gfCNCPoint1[1221] = {X 523.1434, Y 21.1314, Z -1.3333, A 0.000, B 0.000, C 0.000 }
gfCNCPoint1[1222] = {X 523.9777, Y 20.6072, Z -1.3333, A 0.000, B 0.000, C 0.000 }
gfCNCPoint1[1223] = {X 524.9077, Y 20.2817, Z -1.3333, A 0.000, B 0.000, C 0.000 }
gfCNCPoint1[1224] = {X 525.8868, Y 20.1714, Z -1.3333, A 0.000, B 0.000, C 0.000 }
gfCNCPoint1[1225] = {X 526.5702, Y 20.1716, Z -1.3333, A 0.000, B 0.000, C 0.000 }
gfCNCPoint1[1226] = {X 527.4025, Y 20.2591, Z -1.3333, A 0.000, B 0.000, C 0.000 }
gfCNCPoint1[1227] = {X 528.2032, Y 20.5026, Z -1.3333, A 0.000, B 0.000, C 0.000 }
gfCNCPoint1[1228] = {X 528.9433, Y 20.8933, Z -1.3333, A 0.000, B 0.000, C 0.000 }
gfCNCPoint1[1229] = {X 529.5960, Y 21.4171, Z -1.3333, A 0.000, B 0.000, C 0.000 }
gfCNCPoint1[1230] = {X 530.1378, Y 22.0550, Z -1.3333, A 0.000, B 0.000, C 0.000 }
gfCNCPoint1[1231] = {X 534.5519, Y 22.0554, Z -1.3333, A 0.000, B 0.000, C 0.000 }
gfCNCPoint1[1232] = {X 534.5519, Y 19.7809, Z -1.3333, A 0.000, B 0.000, C 0.000 }
gfCNCPoint1[1233] = {X 528.8157, Y 19.7807, Z -1.3333, A 0.000, B 0.000, C 0.000 }
gfCNCPoint1[1234] = {X 528.8157, Y 20.2607, Z -1.3333, A 0.000, B 0.000, C 0.000 }
gfCNCPoint1[1235] = {X 534.0719, Y 20.2609, Z -1.3333, A 0.000, B 0.000, C 0.000 }
gfCNCPoint1[1236] = {X 534.0719, Y 21.5753, Z -1.3333, A 0.000, B 0.000, C 0.000 }
gfCNCPoint1[1237] = {X 530.3802, Y 21.5750, Z -1.3333, A 0.000, B 0.000, C 0.000 }
gfCNCPoint1[1238] = {X 529.6675, Y 20.8350, Z -1.3333, A 0.000, B 0.000, C 0.000 }
gfCNCPoint1[1239] = {X 528.8157, Y 20.2607, Z -1.3333, A 0.000, B 0.000, C 0.000 }
gfCNCPoint1[1240] = {X 528.8157, Y 19.7807, Z -1.3333, A 0.000, B 0.000, C 0.000 }
gfCNCPoint1[1241] = {X 524.2352, Y 19.7804, Z -1.3333, A 0.000, B 0.000, C 0.000 }
gfCNCPoint1[1242] = {X 523.6875, Y 20.4311, Z -1.3333, A 0.000, B 0.000, C 0.000 }
gfCNCPoint1[1243] = {X 523.0249, Y 20.9643, Z -1.3333, A 0.000, B 0.000, C 0.000 }
gfCNCPoint1[1244] = {X 522.2721, Y 21.3600, Z -1.3333, A 0.000, B 0.000, C 0.000 }
gfCNCPoint1[1245] = {X 521.4572, Y 21.6035, Z -1.3333, A 0.000, B 0.000, C 0.000 }
gfCNCPoint1[1246] = {X 520.6107, Y 21.6857, Z -1.3333, A 0.000, B 0.000, C 0.000 }
gfCNCPoint1[1247] = {X 519.9691, Y 21.6857, Z -1.3333, A 0.000, B 0.000, C 0.000 }
gfCNCPoint1[1248] = {X 518.9900, Y 21.5754, Z -1.3333, A 0.000, B 0.000, C 0.000 }
gfCNCPoint1[1249] = {X 518.0600, Y 21.2500, Z -1.3333, A 0.000, B 0.000, C 0.000 }
gfCNCPoint1[1250] = {X 517.2257, Y 20.7258, Z -1.3333, A 0.000, B 0.000, C 0.000 }
gfCNCPoint1[1251] = {X 516.5290, Y 20.0291, Z -1.3333, A 0.000, B 0.000, C 0.000 }
gfCNCPoint1[1252] = {X 516.0048, Y 19.1948, Z -1.3333, A 0.000, B 0.000, C 0.000 }
gfCNCPoint1[1253] = {X 515.6794, Y 18.2648, Z -1.3333, A 0.000, B 0.000, C 0.000 }
gfCNCPoint1[1254] = {X 515.5691, Y 17.2857, Z -1.3333, A 0.000, B 0.000, C 0.000 }
gfCNCPoint1[1255] = {X 515.5691, Y 10.3077, Z -1.3333, A 0.000, B 0.000, C 0.000 }
gfCNCPoint1[1256] = {X 515.6394, Y 9.5244, Z -1.3333, A 0.000, B 0.000, C 0.000 }
gfCNCPoint1[1257] = {X 515.8480, Y 8.7662, Z -1.3333, A 0.000, B 0.000, C 0.000 }
gfCNCPoint1[1258] = {X 516.1882, Y 8.0572, Z -1.3333, A 0.000, B 0.000, C 0.000 }
gfCNCPoint1[1259] = {X 516.6492, Y 7.4201, Z -1.3333, A 0.000, B 0.000, C 0.000 }
gfCNCPoint1[1260] = {X 516.2870, Y 7.1051, Z -1.3333, A 0.000, B 0.000, C 0.000 }
gfCNCPoint1[1261] = {X 469.2627, Y 7.1051, Z -1.3333, A 0.000, B 0.000, C 0.000 }
gfCNCPoint1[1262] = {X 469.2627, Y 11.9051, Z -1.3333, A 0.000, B 0.000, C 0.000 }
gfCNCPoint1[1263] = {X 469.1139, Y 11.9051, Z -1.3333, A 0.000, B 0.000, C 0.000 }
gfCNCPoint1[1264] = {X 469.1170, Y 12.0458, Z -1.3333, A 0.000, B 0.000, C 0.000 }
gfCNCPoint1[1265] = {X 469.1179, Y 12.1865, Z -1.3333, A 0.000, B 0.000, C 0.000 }
gfCNCPoint1[1266] = {X 469.1897, Y 12.0455, Z -1.3333, A 0.000, B 0.000, C 0.000 }
gfCNCPoint1[1267] = {X 469.2627, Y 11.9051, Z -1.3333, A 0.000, B 0.000, C 0.000 }
gfCNCPoint1[1268] = {X 469.2627, Y 9.5051, Z -1.3333, A 0.000, B 0.000, C 0.000 }
gfCNCPoint1[1269] = {X 466.2067, Y 9.5051, Z -1.3333, A 0.000, B 0.000, C 0.000 }
gfCNCPoint1[1270] = {X 466.5686, Y 10.7174, Z -1.3333, A 0.000, B 0.000, C 0.000 }
gfCNCPoint1[1271] = {X 466.7149, Y 11.9742, Z -1.3333, A 0.000, B 0.000, C 0.000 }
gfCNCPoint1[1272] = {X 466.7172, Y 12.0787, Z -1.3333, A 0.000, B 0.000, C 0.000 }
gfCNCPoint1[1273] = {X 466.7179, Y 12.1834, Z -1.3333, A 0.000, B 0.000, C 0.000 }
gfCNCPoint1[1274] = {X 466.7179, Y 12.9779, Z -1.3333, A 0.000, B 0.000, C 0.000 }
gfCNCPoint1[1275] = {X 466.6191, Y 14.1735, Z -1.3333, A 0.000, B 0.000, C 0.000 }
gfCNCPoint1[1276] = {X 466.3252, Y 15.3367, Z -1.3333, A 0.000, B 0.000, C 0.000 }
gfCNCPoint1[1277] = {X 465.8443, Y 16.4358, Z -1.3333, A 0.000, B 0.000, C 0.000 }
gfCNCPoint1[1278] = {X 465.1894, Y 17.4410, Z -1.3333, A 0.000, B 0.000, C 0.000 }
gfCNCPoint1[1279] = {X 465.1896, Y 25.8683, Z -1.3333, A 0.000, B 0.000, C 0.000 }
gfCNCPoint1[1280] = {X 467.5896, Y 25.8683, Z -1.3333, A 0.000, B 0.000, C 0.000 }
gfCNCPoint1[1281] = {X 467.5898, Y 38.9887, Z -1.3333, A 0.000, B 0.000, C 0.000 }
gfCNCPoint1[1282] = {X 467.6015, Y 39.0069, Z -1.3333, A 0.000, B 0.000, C 0.000 }
gfCNCPoint1[1283] = {X 468.3506, Y 37.9855, Z -1.3333, A 0.000, B 0.000, C 0.000 }
gfCNCPoint1[1284] = {X 469.2267, Y 37.0706, Z -1.3333, A 0.000, B 0.000, C 0.000 }
gfCNCPoint1[1285] = {X 470.2148, Y 36.2780, Z -1.3333, A 0.000, B 0.000, C 0.000 }
gfCNCPoint1[1286] = {X 471.5281, Y 33.7072, Z -1.3333, A 0.000, B 0.000, C 0.000 }
gfCNCPoint1[1287] = {X 470.4815, Y 32.4113, Z -1.3333, A 0.000, B 0.000, C 0.000 }
gfCNCPoint1[1288] = {X 469.5681, Y 31.0183, Z -1.3333, A 0.000, B 0.000, C 0.000 }
gfCNCPoint1[1289] = {X 468.7969, Y 29.5419, Z -1.3333, A 0.000, B 0.000, C 0.000 }
gfCNCPoint1[1290] = {X 468.1754, Y 27.9964, Z -1.3333, A 0.000, B 0.000, C 0.000 }
gfCNCPoint1[1291] = {X 467.7096, Y 26.3971, Z -1.3333, A 0.000, B 0.000, C 0.000 }
gfCNCPoint1[1292] = {X 467.6480, Y 26.1331, Z -1.3333, A 0.000, B 0.000, C 0.000 }
gfCNCPoint1[1293] = {X 467.5896, Y 25.8683, Z -1.3333, A 0.000, B 0.000, C 0.000 }
gfCNCPoint1[1294] = {X 465.1896, Y 25.8683, Z -1.3333, A 0.000, B 0.000, C 0.000 }
gfCNCPoint1[1295] = {X 465.1898, Y 39.7463, Z -1.3333, A 0.000, B 0.000, C 0.000 }
gfCNCPoint1[1296] = {X 465.3900, Y 40.0170, Z -1.3333, A 0.000, B 0.000, C 0.000 }
gfCNCPoint1[1297] = {X 465.5774, Y 40.2966, Z -1.3333, A 0.000, B 0.000, C 0.000 }
gfCNCPoint1[1298] = {X 466.0634, Y 41.1919, Z -1.3333, A 0.000, B 0.000, C 0.000 }
gfCNCPoint1[1299] = {X 466.4196, Y 42.1462, Z -1.3333, A 0.000, B 0.000, C 0.000 }
gfCNCPoint1[1300] = {X 466.6392, Y 43.1408, Z -1.3333, A 0.000, B 0.000, C 0.000 }
gfCNCPoint1[1301] = {X 466.7178, Y 44.1564, Z -1.3333, A 0.000, B 0.000, C 0.000 }
gfCNCPoint1[1302] = {X 466.7179, Y 45.0000, Z -1.3333, A 0.000, B 0.000, C 0.000 }
gfCNCPoint1[1303] = {X 466.7033, Y 45.4609, Z -1.3333, A 0.000, B 0.000, C 0.000 }
gfCNCPoint1[1304] = {X 466.6596, Y 45.9200, Z -1.3333, A 0.000, B 0.000, C 0.000 }
gfCNCPoint1[1305] = {X 468.5433, Y 45.9200, Z -1.3333, A 0.000, B 0.000, C 0.000 }
gfCNCPoint1[1306] = {X 468.4996, Y 45.4609, Z -1.3333, A 0.000, B 0.000, C 0.000 }
gfCNCPoint1[1307] = {X 468.4850, Y 45.0000, Z -1.3333, A 0.000, B 0.000, C 0.000 }
gfCNCPoint1[1308] = {X 468.4850, Y 44.2090, Z -1.3333, A 0.000, B 0.000, C 0.000 }
gfCNCPoint1[1309] = {X 468.5580, Y 43.1799, Z -1.3333, A 0.000, B 0.000, C 0.000 }
gfCNCPoint1[1310] = {X 468.7759, Y 42.1714, Z -1.3333, A 0.000, B 0.000, C 0.000 }
gfCNCPoint1[1311] = {X 469.1341, Y 41.2038, Z -1.3333, A 0.000, B 0.000, C 0.000 }
gfCNCPoint1[1312] = {X 469.6255, Y 40.2966, Z -1.3333, A 0.000, B 0.000, C 0.000 }
gfCNCPoint1[1313] = {X 470.3102, Y 39.3876, Z -1.3333, A 0.000, B 0.000, C 0.000 }
gfCNCPoint1[1314] = {X 471.1282, Y 38.5964, Z -1.3333, A 0.000, B 0.000, C 0.000 }
gfCNCPoint1[1315] = {X 472.0595, Y 37.9424, Z -1.3333, A 0.000, B 0.000, C 0.000 }
gfCNCPoint1[1316] = {X 474.4573, Y 33.2490, Z -1.3333, A 0.000, B 0.000, C 0.000 }
gfCNCPoint1[1317] = {X 473.2262, Y 32.0044, Z -1.3333, A 0.000, B 0.000, C 0.000 }
gfCNCPoint1[1318] = {X 472.1548, Y 30.6199, Z -1.3333, A 0.000, B 0.000, C 0.000 }
gfCNCPoint1[1319] = {X 471.2590, Y 29.1158, Z -1.3333, A 0.000, B 0.000, C 0.000 }
gfCNCPoint1[1320] = {X 470.5519, Y 27.5144, Z -1.3333, A 0.000, B 0.000, C 0.000 }
gfCNCPoint1[1321] = {X 470.0438, Y 25.8391, Z -1.3333, A 0.000, B 0.000, C 0.000 }
gfCNCPoint1[1322] = {X 469.9887, Y 25.6028, Z -1.3333, A 0.000, B 0.000, C 0.000 }
gfCNCPoint1[1323] = {X 469.9364, Y 25.3658, Z -1.3333, A 0.000, B 0.000, C 0.000 }
gfCNCPoint1[1324] = {X 469.6267, Y 23.4734, Z -1.3333, A 0.000, B 0.000, C 0.000 }
gfCNCPoint1[1325] = {X 469.5026, Y 21.5599, Z -1.3333, A 0.000, B 0.000, C 0.000 }
gfCNCPoint1[1326] = {X 469.5653, Y 19.6434, Z -1.3333, A 0.000, B 0.000, C 0.000 }
gfCNCPoint1[1327] = {X 469.8141, Y 17.7420, Z -1.3333, A 0.000, B 0.000, C 0.000 }
gfCNCPoint1[1328] = {X 470.2468, Y 15.8739, Z -1.3333, A 0.000, B 0.000, C 0.000 }
gfCNCPoint1[1329] = {X 470.6926, Y 14.5452, Z -1.3333, A 0.000, B 0.000, C 0.000 }
gfCNCPoint1[1330] = {X 471.2622, Y 13.2646, Z -1.3333, A 0.000, B 0.000, C 0.000 }
gfCNCPoint1[1331] = {X 471.3239, Y 13.1432, Z -1.3333, A 0.000, B 0.000, C 0.000 }
gfCNCPoint1[1332] = {X 471.3867, Y 13.0225, Z -1.3333, A 0.000, B 0.000, C 0.000 }
gfCNCPoint1[1333] = {X 472.1282, Y 11.7671, Z -1.3333, A 0.000, B 0.000, C 0.000 }
gfCNCPoint1[1334] = {X 472.9897, Y 10.5909, Z -1.3333, A 0.000, B 0.000, C 0.000 }
gfCNCPoint1[1335] = {X 473.9628, Y 9.5051, Z -1.3333, A 0.000, B 0.000, C 0.000 }
gfCNCPoint1[1336] = {X 469.2627, Y 9.5051, Z -1.3333, A 0.000, B 0.000, C 0.000 }
gfCNCPoint1[1337] = {X 469.2627, Y 7.1051, Z -1.3333, A 0.000, B 0.000, C 0.000 }
gfCNCPoint1[1338] = {X 370.1016, Y 7.1051, Z -1.3333, A 0.000, B 0.000, C 0.000 }
gfCNCPoint1[1339] = {X 371.1252, Y 8.7921, Z -1.3333, A 0.000, B 0.000, C 0.000 }
gfCNCPoint1[1340] = {X 372.0361, Y 10.5425, Z -1.3333, A 0.000, B 0.000, C 0.000 }
gfCNCPoint1[1341] = {X 372.9332, Y 12.6093, Z -1.3333, A 0.000, B 0.000, C 0.000 }
gfCNCPoint1[1342] = {X 373.6731, Y 14.7374, Z -1.3333, A 0.000, B 0.000, C 0.000 }
gfCNCPoint1[1343] = {X 374.2517, Y 16.9150, Z -1.3333, A 0.000, B 0.000, C 0.000 }
gfCNCPoint1[1344] = {X 374.7361, Y 19.4755, Z -1.3333, A 0.000, B 0.000, C 0.000 }
gfCNCPoint1[1345] = {X 375.0392, Y 22.0637, Z -1.3333, A 0.000, B 0.000, C 0.000 }
gfCNCPoint1[1346] = {X 375.1593, Y 24.6669, Z -1.3333, A 0.000, B 0.000, C 0.000 }
gfCNCPoint1[1347] = {X 375.0959, Y 27.2721, Z -1.3333, A 0.000, B 0.000, C 0.000 }
gfCNCPoint1[1348] = {X 374.8493, Y 29.8664, Z -1.3333, A 0.000, B 0.000, C 0.000 }
gfCNCPoint1[1349] = {X 374.4207, Y 32.4368, Z -1.3333, A 0.000, B 0.000, C 0.000 }
gfCNCPoint1[1350] = {X 373.7829, Y 34.9988, Z -1.3333, A 0.000, B 0.000, C 0.000 }
gfCNCPoint1[1351] = {X 372.9214, Y 37.4945, Z -1.3333, A 0.000, B 0.000, C 0.000 }
gfCNCPoint1[1352] = {X 371.8430, Y 39.9043, Z -1.3333, A 0.000, B 0.000, C 0.000 }
gfCNCPoint1[1353] = {X 370.5559, Y 42.2095, Z -1.3333, A 0.000, B 0.000, C 0.000 }
gfCNCPoint1[1354] = {X 369.0704, Y 44.3921, Z -1.3333, A 0.000, B 0.000, C 0.000 }
gfCNCPoint1[1355] = {X 369.0316, Y 44.4442, Z -1.3333, A 0.000, B 0.000, C 0.000 }
gfCNCPoint1[1356] = {X 368.9927, Y 44.4963, Z -1.3333, A 0.000, B 0.000, C 0.000 }
gfCNCPoint1[1357] = {X 367.4727, Y 46.3512, Z -1.3333, A 0.000, B 0.000, C 0.000 }
gfCNCPoint1[1358] = {X 365.7972, Y 48.0668, Z -1.3333, A 0.000, B 0.000, C 0.000 }
gfCNCPoint1[1359] = {X 363.9787, Y 49.6301, Z -1.3333, A 0.000, B 0.000, C 0.000 }
gfCNCPoint1[1360] = {X 362.0311, Y 51.0293, Z -1.3333, A 0.000, B 0.000, C 0.000 }
gfCNCPoint1[1361] = {X 359.9692, Y 52.2538, Z -1.3333, A 0.000, B 0.000, C 0.000 }
gfCNCPoint1[1362] = {X 359.3965, Y 52.5409, Z -1.3333, A 0.000, B 0.000, C 0.000 }
gfCNCPoint1[1363] = {X 358.8175, Y 52.8148, Z -1.3333, A 0.000, B 0.000, C 0.000 }
gfCNCPoint1[1364] = {X 356.4598, Y 53.7700, Z -1.3333, A 0.000, B 0.000, C 0.000 }
gfCNCPoint1[1365] = {X 354.0251, Y 54.5072, Z -1.3333, A 0.000, B 0.000, C 0.000 }
gfCNCPoint1[1366] = {X 351.5336, Y 55.0204, Z -1.3333, A 0.000, B 0.000, C 0.000 }
gfCNCPoint1[1367] = {X 349.0058, Y 55.3053, Z -1.3333, A 0.000, B 0.000, C 0.000 }
gfCNCPoint1[1368] = {X 349.9666, Y 69.6732, Z -1.3333, A 0.000, B 0.000, C 0.000 }
gfCNCPoint1[1369] = {X 348.6526, Y 69.7406, Z -1.3333, A 0.000, B 0.000, C 0.000 }
gfCNCPoint1[1370] = {X 347.3372, Y 69.7672, Z -1.3333, A 0.000, B 0.000, C 0.000 }
gfCNCPoint1[1371] = {X 346.5718, Y 69.7758, Z -1.3333, A 0.000, B 0.000, C 0.000 }
gfCNCPoint1[1372] = {X 345.8063, Y 69.7711, Z -1.3333, A 0.000, B 0.000, C 0.000 }
gfCNCPoint1[1373] = {X 345.5910, Y 70.1878, Z -1.3333, A 0.000, B 0.000, C 0.000 }
gfCNCPoint1[1374] = {X 345.3676, Y 70.6003, Z -1.3333, A 0.000, B 0.000, C 0.000 }
gfCNCPoint1[1375] = {X 345.9399, Y 70.6040, Z -1.3333, A 0.000, B 0.000, C 0.000 }
gfCNCPoint1[1376] = {X 348.1990, Y 70.6282, Z -1.3333, A 0.000, B 0.000, C 0.000 }
gfCNCPoint1[1377] = {X 350.4581, Y 70.6078, Z -1.3333, A 0.000, B 0.000, C 0.000 }
gfCNCPoint1[1378] = {X 350.2072, Y 70.1432, Z -1.3333, A 0.000, B 0.000, C 0.000 }
gfCNCPoint1[1379] = {X 349.9666, Y 69.6732, Z -1.3333, A 0.000, B 0.000, C 0.000 }
gfCNCPoint1[1380] = {X 349.8065, Y 67.2785, Z -1.3333, A 0.000, B 0.000, C 0.000 }
gfCNCPoint1[1381] = {X 348.5577, Y 67.3424, Z -1.3333, A 0.000, B 0.000, C 0.000 }
gfCNCPoint1[1382] = {X 347.3075, Y 67.3673, Z -1.3333, A 0.000, B 0.000, C 0.000 }
gfCNCPoint1[1383] = {X 345.8014, Y 67.3707, Z -1.3333, A 0.000, B 0.000, C 0.000 }
gfCNCPoint1[1384] = {X 344.2963, Y 67.3191, Z -1.3333, A 0.000, B 0.000, C 0.000 }
gfCNCPoint1[1385] = {X 343.8111, Y 68.3919, Z -1.3333, A 0.000, B 0.000, C 0.000 }
gfCNCPoint1[1386] = {X 343.2685, Y 69.4370, Z -1.3333, A 0.000, B 0.000, C 0.000 }
gfCNCPoint1[1387] = {X 342.7876, Y 70.2613, Z -1.3333, A 0.000, B 0.000, C 0.000 }
gfCNCPoint1[1388] = {X 342.2711, Y 71.0637, Z -1.3333, A 0.000, B 0.000, C 0.000 }
gfCNCPoint1[1389] = {X 342.2712, Y 72.9213, Z -1.3333, A 0.000, B 0.000, C 0.000 }
gfCNCPoint1[1390] = {X 343.8076, Y 72.9731, Z -1.3333, A 0.000, B 0.000, C 0.000 }
gfCNCPoint1[1391] = {X 345.3447, Y 73.0002, Z -1.3333, A 0.000, B 0.000, C 0.000 }
gfCNCPoint1[1392] = {X 345.6279, Y 73.0025, Z -1.3333, A 0.000, B 0.000, C 0.000 }
gfCNCPoint1[1393] = {X 345.9111, Y 73.0039, Z -1.3333, A 0.000, B 0.000, C 0.000 }
gfCNCPoint1[1394] = {X 348.2072, Y 73.0282, Z -1.3333, A 0.000, B 0.000, C 0.000 }
gfCNCPoint1[1395] = {X 350.5035, Y 73.0073, Z -1.3333, A 0.000, B 0.000, C 0.000 }
gfCNCPoint1[1396] = {X 352.0323, Y 72.9685, Z -1.3333, A 0.000, B 0.000, C 0.000 }
gfCNCPoint1[1397] = {X 353.5605, Y 72.9096, Z -1.3333, A 0.000, B 0.000, C 0.000 }
gfCNCPoint1[1398] = {X 353.5603, Y 71.0790, Z -1.3333, A 0.000, B 0.000, C 0.000 }
gfCNCPoint1[1399] = {X 353.0407, Y 70.2727, Z -1.3333, A 0.000, B 0.000, C 0.000 }
gfCNCPoint1[1400] = {X 352.5573, Y 69.4443, Z -1.3333, A 0.000, B 0.000, C 0.000 }
gfCNCPoint1[1401] = {X 351.9695, Y 68.3058, Z -1.3333, A 0.000, B 0.000, C 0.000 }
gfCNCPoint1[1402] = {X 351.4500, Y 67.1345, Z -1.3333, A 0.000, B 0.000, C 0.000 }
gfCNCPoint1[1403] = {X 350.6290, Y 67.2150, Z -1.3333, A 0.000, B 0.000, C 0.000 }
gfCNCPoint1[1404] = {X 349.8065, Y 67.2785, Z -1.3333, A 0.000, B 0.000, C 0.000 }
gfCNCPoint1[1405] = {X 349.6463, Y 64.8839, Z -1.3333, A 0.000, B 0.000, C 0.000 }
gfCNCPoint1[1406] = {X 348.4627, Y 64.9443, Z -1.3333, A 0.000, B 0.000, C 0.000 }
gfCNCPoint1[1407] = {X 347.2777, Y 64.9674, Z -1.3333, A 0.000, B 0.000, C 0.000 }
gfCNCPoint1[1408] = {X 344.9730, Y 64.9474, Z -1.3333, A 0.000, B 0.000, C 0.000 }
gfCNCPoint1[1409] = {X 342.6736, Y 64.7906, Z -1.3333, A 0.000, B 0.000, C 0.000 }
gfCNCPoint1[1410] = {X 341.9387, Y 66.7258, Z -1.3333, A 0.000, B 0.000, C 0.000 }
gfCNCPoint1[1411] = {X 341.0009, Y 68.5712, Z -1.3333, A 0.000, B 0.000, C 0.000 }
gfCNCPoint1[1412] = {X 339.8710, Y 70.3057, Z -1.3333, A 0.000, B 0.000, C 0.000 }
gfCNCPoint1[1413] = {X 339.8714, Y 75.1959, Z -1.3333, A 0.000, B 0.000, C 0.000 }
gfCNCPoint1[1414] = {X 342.8752, Y 75.3461, Z -1.3333, A 0.000, B 0.000, C 0.000 }
gfCNCPoint1[1415] = {X 345.8822, Y 75.4038, Z -1.3333, A 0.000, B 0.000, C 0.000 }
gfCNCPoint1[1416] = {X 350.9238, Y 75.3992, Z -1.3333, A 0.000, B 0.000, C 0.000 }
gfCNCPoint1[1417] = {X 355.9607, Y 75.1818, Z -1.3333, A 0.000, B 0.000, C 0.000 }
gfCNCPoint1[1418] = {X 355.9603, Y 70.3198, Z -1.3333, A 0.000, B 0.000, C 0.000 }
gfCNCPoint1[1419] = {X 355.0524, Y 68.9620, Z -1.3333, A 0.000, B 0.000, C 0.000 }
gfCNCPoint1[1420] = {X 354.2627, Y 67.5323, Z -1.3333, A 0.000, B 0.000, C 0.000 }
gfCNCPoint1[1421] = {X 353.5969, Y 66.0408, Z -1.3333, A 0.000, B 0.000, C 0.000 }
gfCNCPoint1[1422] = {X 353.0597, Y 64.4983, Z -1.3333, A 0.000, B 0.000, C 0.000 }
gfCNCPoint1[1423] = {X 351.3574, Y 64.7301, Z -1.3333, A 0.000, B 0.000, C 0.000 }
gfCNCPoint1[1424] = {X 349.6463, Y 64.8839, Z -1.3333, A 0.000, B 0.000, C 0.000 }
gfCNCPoint1[1425] = {X 349.4862, Y 62.4892, Z -1.3333, A 0.000, B 0.000, C 0.000 }
gfCNCPoint1[1426] = {X 348.3677, Y 62.5461, Z -1.3333, A 0.000, B 0.000, C 0.000 }
gfCNCPoint1[1427] = {X 347.2480, Y 62.5675, Z -1.3333, A 0.000, B 0.000, C 0.000 }
gfCNCPoint1[1428] = {X 345.1177, Y 62.5512, Z -1.3333, A 0.000, B 0.000, C 0.000 }
gfCNCPoint1[1429] = {X 342.9921, Y 62.4102, Z -1.3333, A 0.000, B 0.000, C 0.000 }
gfCNCPoint1[1430] = {X 340.8784, Y 62.1450, Z -1.3333, A 0.000, B 0.000, C 0.000 }
gfCNCPoint1[1431] = {X 340.4884, Y 63.7331, Z -1.3333, A 0.000, B 0.000, C 0.000 }
gfCNCPoint1[1432] = {X 339.9469, Y 65.2761, Z -1.3333, A 0.000, B 0.000, C 0.000 }
gfCNCPoint1[1433] = {X 339.2590, Y 66.7596, Z -1.3333, A 0.000, B 0.000, C 0.000 }
gfCNCPoint1[1434] = {X 338.4311, Y 68.1698, Z -1.3333, A 0.000, B 0.000, C 0.000 }
gfCNCPoint1[1435] = {X 337.4710, Y 69.4935, Z -1.3333, A 0.000, B 0.000, C 0.000 }
gfCNCPoint1[1436] = {X 337.4715, Y 77.4188, Z -1.3333, A 0.000, B 0.000, C 0.000 }
gfCNCPoint1[1437] = {X 341.6584, Y 77.6990, Z -1.3333, A 0.000, B 0.000, C 0.000 }
gfCNCPoint1[1438] = {X 345.8533, Y 77.8037, Z -1.3333, A 0.000, B 0.000, C 0.000 }
gfCNCPoint1[1439] = {X 350.0262, Y 77.8159, Z -1.3333, A 0.000, B 0.000, C 0.000 }
gfCNCPoint1[1440] = {X 354.1970, Y 77.6851, Z -1.3333, A 0.000, B 0.000, C 0.000 }
gfCNCPoint1[1441] = {X 358.3609, Y 77.4115, Z -1.3333, A 0.000, B 0.000, C 0.000 }
gfCNCPoint1[1442] = {X 358.3602, Y 69.5063, Z -1.3333, A 0.000, B 0.000, C 0.000 }
gfCNCPoint1[1443] = {X 357.3489, Y 68.1066, Z -1.3333, A 0.000, B 0.000, C 0.000 }
gfCNCPoint1[1444] = {X 356.4859, Y 66.6108, Z -1.3333, A 0.000, B 0.000, C 0.000 }
gfCNCPoint1[1445] = {X 355.7802, Y 65.0347, Z -1.3333, A 0.000, B 0.000, C 0.000 }
gfCNCPoint1[1446] = {X 355.2393, Y 63.3947, Z -1.3333, A 0.000, B 0.000, C 0.000 }
gfCNCPoint1[1447] = {X 354.8688, Y 61.7081, Z -1.3333, A 0.000, B 0.000, C 0.000 }
gfCNCPoint1[1448] = {X 352.1926, Y 62.2028, Z -1.3333, A 0.000, B 0.000, C 0.000 }
gfCNCPoint1[1449] = {X 349.4862, Y 62.4892, Z -1.3333, A 0.000, B 0.000, C 0.000 }
gfCNCPoint1[1450] = {X 349.3260, Y 60.0946, Z -1.3333, A 0.000, B 0.000, C 0.000 }
gfCNCPoint1[1451] = {X 348.2727, Y 60.1480, Z -1.3333, A 0.000, B 0.000, C 0.000 }
gfCNCPoint1[1452] = {X 347.2182, Y 60.1675, Z -1.3333, A 0.000, B 0.000, C 0.000 }
gfCNCPoint1[1453] = {X 344.3864, Y 60.1126, Z -1.3333, A 0.000, B 0.000, C 0.000 }
gfCNCPoint1[1454] = {X 341.5690, Y 59.8219, Z -1.3333, A 0.000, B 0.000, C 0.000 }
gfCNCPoint1[1455] = {X 338.7855, Y 59.2975, Z -1.3333, A 0.000, B 0.000, C 0.000 }
gfCNCPoint1[1456] = {X 338.6398, Y 60.9970, Z -1.3333, A 0.000, B 0.000, C 0.000 }
gfCNCPoint1[1457] = {X 338.2957, Y 62.6677, Z -1.3333, A 0.000, B 0.000, C 0.000 }
gfCNCPoint1[1458] = {X 337.7581, Y 64.2865, Z -1.3333, A 0.000, B 0.000, C 0.000 }
gfCNCPoint1[1459] = {X 337.0344, Y 65.8310, Z -1.3333, A 0.000, B 0.000, C 0.000 }
gfCNCPoint1[1460] = {X 336.1345, Y 67.2801, Z -1.3333, A 0.000, B 0.000, C 0.000 }
gfCNCPoint1[1461] = {X 335.0709, Y 68.6136, Z -1.3333, A 0.000, B 0.000, C 0.000 }
gfCNCPoint1[1462] = {X 335.0717, Y 79.5892, Z -1.3333, A 0.000, B 0.000, C 0.000 }
gfCNCPoint1[1463] = {X 335.6784, Y 79.6597, Z -1.3333, A 0.000, B 0.000, C 0.000 }
gfCNCPoint1[1464] = {X 336.2864, Y 79.7191, Z -1.3333, A 0.000, B 0.000, C 0.000 }
gfCNCPoint1[1465] = {X 341.0497, Y 80.0723, Z -1.3333, A 0.000, B 0.000, C 0.000 }
gfCNCPoint1[1466] = {X 345.8244, Y 80.2036, Z -1.3333, A 0.000, B 0.000, C 0.000 }
gfCNCPoint1[1467] = {X 350.3389, Y 80.2114, Z -1.3333, A 0.000, B 0.000, C 0.000 }
gfCNCPoint1[1468] = {X 354.8507, Y 80.0550, Z -1.3333, A 0.000, B 0.000, C 0.000 }
gfCNCPoint1[1469] = {X 359.3538, Y 79.7348, Z -1.3333, A 0.000, B 0.000, C 0.000 }
gfCNCPoint1[1470] = {X 360.0583, Y 79.6699, Z -1.3333, A 0.000, B 0.000, C 0.000 }
gfCNCPoint1[1471] = {X 360.7611, Y 79.5886, Z -1.3333, A 0.000, B 0.000, C 0.000 }
gfCNCPoint1[1472] = {X 360.7601, Y 68.6248, Z -1.3333, A 0.000, B 0.000, C 0.000 }
gfCNCPoint1[1473] = {X 359.7308, Y 67.3425, Z -1.3333, A 0.000, B 0.000, C 0.000 }
gfCNCPoint1[1474] = {X 358.8534, Y 65.9517, Z -1.3333, A 0.000, B 0.000, C 0.000 }
gfCNCPoint1[1475] = {X 358.1395, Y 64.4704, Z -1.3333, A 0.000, B 0.000, C 0.000 }
gfCNCPoint1[1476] = {X 357.5980, Y 62.9177, Z -1.3333, A 0.000, B 0.000, C 0.000 }
gfCNCPoint1[1477] = {X 357.2361, Y 61.3136, Z -1.3333, A 0.000, B 0.000, C 0.000 }
gfCNCPoint1[1478] = {X 357.0916, Y 60.1644, Z -1.3333, A 0.000, B 0.000, C 0.000 }
gfCNCPoint1[1479] = {X 357.0395, Y 59.0073, Z -1.3333, A 0.000, B 0.000, C 0.000 }
gfCNCPoint1[1480] = {X 357.0394, Y 58.6372, Z -1.3333, A 0.000, B 0.000, C 0.000 }
gfCNCPoint1[1481] = {X 355.6983, Y 59.0307, Z -1.3333, A 0.000, B 0.000, C 0.000 }
gfCNCPoint1[1482] = {X 354.3416, Y 59.3667, Z -1.3333, A 0.000, B 0.000, C 0.000 }
gfCNCPoint1[1483] = {X 351.8479, Y 59.8276, Z -1.3333, A 0.000, B 0.000, C 0.000 }
gfCNCPoint1[1484] = {X 349.3260, Y 60.0946, Z -1.3333, A 0.000, B 0.000, C 0.000 }
gfCNCPoint1[1485] = {X 349.1659, Y 57.6999, Z -1.3333, A 0.000, B 0.000, C 0.000 }
gfCNCPoint1[1486] = {X 348.1778, Y 57.7498, Z -1.3333, A 0.000, B 0.000, C 0.000 }
gfCNCPoint1[1487] = {X 347.1886, Y 57.7676, Z -1.3333, A 0.000, B 0.000, C 0.000 }
gfCNCPoint1[1488] = {X 344.5488, Y 57.7180, Z -1.3333, A 0.000, B 0.000, C 0.000 }
gfCNCPoint1[1489] = {X 341.9225, Y 57.4481, Z -1.3333, A 0.000, B 0.000, C 0.000 }
gfCNCPoint1[1490] = {X 339.3279, Y 56.9596, Z -1.3333, A 0.000, B 0.000, C 0.000 }
gfCNCPoint1[1491] = {X 337.7707, Y 56.5563, Z -1.3333, A 0.000, B 0.000, C 0.000 }
gfCNCPoint1[1492] = {X 336.2362, Y 56.0743, Z -1.3333, A 0.000, B 0.000, C 0.000 }
gfCNCPoint1[1493] = {X 336.3520, Y 57.0340, Z -1.3333, A 0.000, B 0.000, C 0.000 }
gfCNCPoint1[1494] = {X 336.3907, Y 58.0000, Z -1.3333, A 0.000, B 0.000, C 0.000 }
gfCNCPoint1[1495] = {X 336.3907, Y 58.9501, Z -1.3333, A 0.000, B 0.000, C 0.000 }
gfCNCPoint1[1496] = {X 336.3894, Y 59.0917, Z -1.3333, A 0.000, B 0.000, C 0.000 }
gfCNCPoint1[1497] = {X 336.3864, Y 59.2332, Z -1.3333, A 0.000, B 0.000, C 0.000 }
gfCNCPoint1[1498] = {X 336.2426, Y 60.7976, Z -1.3333, A 0.000, B 0.000, C 0.000 }
gfCNCPoint1[1499] = {X 335.8977, Y 62.3303, Z -1.3333, A 0.000, B 0.000, C 0.000 }
gfCNCPoint1[1500] = {X 335.3575, Y 63.8054, Z -1.3333, A 0.000, B 0.000, C 0.000 }
gfCNCPoint1[1501] = {X 334.6310, Y 65.1983, Z -1.3333, A 0.000, B 0.000, C 0.000 }
gfCNCPoint1[1502] = {X 333.7304, Y 66.4856, Z -1.3333, A 0.000, B 0.000, C 0.000 }
gfCNCPoint1[1503] = {X 332.6709, Y 67.6455, Z -1.3333, A 0.000, B 0.000, C 0.000 }
gfCNCPoint1[1504] = {X 332.6718, Y 81.6429, Z -1.3333, A 0.000, B 0.000, C 0.000 }
gfCNCPoint1[1505] = {X 334.3622, Y 81.9165, Z -1.3333, A 0.000, B 0.000, C 0.000 }
gfCNCPoint1[1506] = {X 336.0639, Y 82.1088, Z -1.3333, A 0.000, B 0.000, C 0.000 }
gfCNCPoint1[1507] = {X 340.9239, Y 82.4690, Z -1.3333, A 0.000, B 0.000, C 0.000 }
gfCNCPoint1[1508] = {X 345.7954, Y 82.6035, Z -1.3333, A 0.000, B 0.000, C 0.000 }
gfCNCPoint1[1509] = {X 350.3874, Y 82.6109, Z -1.3333, A 0.000, B 0.000, C 0.000 }
gfCNCPoint1[1510] = {X 354.9766, Y 82.4517, Z -1.3333, A 0.000, B 0.000, C 0.000 }
gfCNCPoint1[1511] = {X 359.5570, Y 82.1262, Z -1.3333, A 0.000, B 0.000, C 0.000 }
gfCNCPoint1[1512] = {X 361.3660, Y 81.9295, Z -1.3333, A 0.000, B 0.000, C 0.000 }
gfCNCPoint1[1513] = {X 363.1612, Y 81.6323, Z -1.3333, A 0.000, B 0.000, C 0.000 }
gfCNCPoint1[1514] = {X 363.1600, Y 67.6547, Z -1.3333, A 0.000, B 0.000, C 0.000 }
gfCNCPoint1[1515] = {X 362.0736, Y 66.4644, Z -1.3333, A 0.000, B 0.000, C 0.000 }
gfCNCPoint1[1516] = {X 361.1553, Y 65.1400, Z -1.3333, A 0.000, B 0.000, C 0.000 }
gfCNCPoint1[1517] = {X 360.4214, Y 63.7052, Z -1.3333, A 0.000, B 0.000, C 0.000 }
gfCNCPoint1[1518] = {X 359.8851, Y 62.1855, Z -1.3333, A 0.000, B 0.000, C 0.000 }
gfCNCPoint1[1519] = {X 359.5558, Y 60.6079, Z -1.3333, A 0.000, B 0.000, C 0.000 }
gfCNCPoint1[1520] = {X 359.4395, Y 59.0005, Z -1.3333, A 0.000, B 0.000, C 0.000 }
gfCNCPoint1[1521] = {X 359.4393, Y 58.0000, Z -1.3333, A 0.000, B 0.000, C 0.000 }
gfCNCPoint1[1522] = {X 359.5345, Y 56.4860, Z -1.3333, A 0.000, B 0.000, C 0.000 }
gfCNCPoint1[1523] = {X 359.8188, Y 54.9959, Z -1.3333, A 0.000, B 0.000, C 0.000 }
gfCNCPoint1[1524] = {X 358.0877, Y 55.7267, Z -1.3333, A 0.000, B 0.000, C 0.000 }
gfCNCPoint1[1525] = {X 356.3148, Y 56.3492, Z -1.3333, A 0.000, B 0.000, C 0.000 }
gfCNCPoint1[1526] = {X 353.9704, Y 56.9897, Z -1.3333, A 0.000, B 0.000, C 0.000 }
gfCNCPoint1[1527] = {X 351.5824, Y 57.4409, Z -1.3333, A 0.000, B 0.000, C 0.000 }
gfCNCPoint1[1528] = {X 349.1659, Y 57.6999, Z -1.3333, A 0.000, B 0.000, C 0.000 }
gfCNCPoint1[1529] = {X 349.0058, Y 55.3053, Z -1.3333, A 0.000, B 0.000, C 0.000 }
gfCNCPoint1[1530] = {X 348.0829, Y 55.3517, Z -1.3333, A 0.000, B 0.000, C 0.000 }
gfCNCPoint1[1531] = {X 347.1589, Y 55.3676, Z -1.3333, A 0.000, B 0.000, C 0.000 }
gfCNCPoint1[1532] = {X 344.5805, Y 55.3153, Z -1.3333, A 0.000, B 0.000, C 0.000 }
gfCNCPoint1[1533] = {X 342.0169, Y 55.0355, Z -1.3333, A 0.000, B 0.000, C 0.000 }
gfCNCPoint1[1534] = {X 339.4880, Y 54.5303, Z -1.3333, A 0.000, B 0.000, C 0.000 }
gfCNCPoint1[1535] = {X 337.0136, Y 53.8037, Z -1.3333, A 0.000, B 0.000, C 0.000 }
gfCNCPoint1[1536] = {X 334.7560, Y 52.9244, Z -1.3333, A 0.000, B 0.000, C 0.000 }
gfCNCPoint1[1537] = {X 332.5792, Y 51.8608, Z -1.3333, A 0.000, B 0.000, C 0.000 }
gfCNCPoint1[1538] = {X 331.5763, Y 51.2697, Z -1.3333, A 0.000, B 0.000, C 0.000 }
gfCNCPoint1[1539] = {X 330.5976, Y 50.6395, Z -1.3333, A 0.000, B 0.000, C 0.000 }
gfCNCPoint1[1540] = {X 331.5681, Y 51.5943, Z -1.3333, A 0.000, B 0.000, C 0.000 }
gfCNCPoint1[1541] = {X 332.3950, Y 52.6759, Z -1.3333, A 0.000, B 0.000, C 0.000 }
gfCNCPoint1[1542] = {X 333.0620, Y 53.8627, Z -1.3333, A 0.000, B 0.000, C 0.000 }
gfCNCPoint1[1543] = {X 333.5559, Y 55.1314, Z -1.3333, A 0.000, B 0.000, C 0.000 }
gfCNCPoint1[1544] = {X 333.8669, Y 56.4569, Z -1.3333, A 0.000, B 0.000, C 0.000 }
gfCNCPoint1[1545] = {X 333.9597, Y 57.2260, Z -1.3333, A 0.000, B 0.000, C 0.000 }
gfCNCPoint1[1546] = {X 333.9907, Y 58.0000, Z -1.3333, A 0.000, B 0.000, C 0.000 }
gfCNCPoint1[1547] = {X 333.9907, Y 58.9455, Z -1.3333, A 0.000, B 0.000, C 0.000 }
gfCNCPoint1[1548] = {X 333.8756, Y 60.4004, Z -1.3333, A 0.000, B 0.000, C 0.000 }
gfCNCPoint1[1549] = {X 333.5440, Y 61.8216, Z -1.3333, A 0.000, B 0.000, C 0.000 }
gfCNCPoint1[1550] = {X 333.0033, Y 63.1772, Z -1.3333, A 0.000, B 0.000, C 0.000 }
gfCNCPoint1[1551] = {X 332.2658, Y 64.4365, Z -1.3333, A 0.000, B 0.000, C 0.000 }
gfCNCPoint1[1552] = {X 331.3481, Y 65.5712, Z -1.3333, A 0.000, B 0.000, C 0.000 }
gfCNCPoint1[1553] = {X 330.2708, Y 66.5557, Z -1.3333, A 0.000, B 0.000, C 0.000 }
gfCNCPoint1[1554] = {X 330.2719, Y 83.2032, Z -1.3333, A 0.000, B 0.000, C 0.000 }
gfCNCPoint1[1555] = {X 330.2756, Y 83.5839, Z -1.3333, A 0.000, B 0.000, C 0.000 }
gfCNCPoint1[1556] = {X 330.3827, Y 83.6094, Z -1.3333, A 0.000, B 0.000, C 0.000 }
gfCNCPoint1[1557] = {X 333.0958, Y 84.1531, Z -1.3333, A 0.000, B 0.000, C 0.000 }
gfCNCPoint1[1558] = {X 335.8411, Y 84.4984, Z -1.3333, A 0.000, B 0.000, C 0.000 }
gfCNCPoint1[1559] = {X 340.7979, Y 84.8657, Z -1.3333, A 0.000, B 0.000, C 0.000 }
gfCNCPoint1[1560] = {X 345.7664, Y 85.0034, Z -1.3333, A 0.000, B 0.000, C 0.000 }
gfCNCPoint1[1561] = {X 350.4359, Y 85.0104, Z -1.3333, A 0.000, B 0.000, C 0.000 }
gfCNCPoint1[1562] = {X 355.1026, Y 84.8484, Z -1.3333, A 0.000, B 0.000, C 0.000 }
gfCNCPoint1[1563] = {X 359.7604, Y 84.5176, Z -1.3333, A 0.000, B 0.000, C 0.000 }
gfCNCPoint1[1564] = {X 361.7111, Y 84.3046, Z -1.3333, A 0.000, B 0.000, C 0.000 }
gfCNCPoint1[1565] = {X 363.6468, Y 83.9829, Z -1.3333, A 0.000, B 0.000, C 0.000 }
gfCNCPoint1[1566] = {X 365.5614, Y 83.5533, Z -1.3333, A 0.000, B 0.000, C 0.000 }
gfCNCPoint1[1567] = {X 365.5599, Y 66.5622, Z -1.3333, A 0.000, B 0.000, C 0.000 }
gfCNCPoint1[1568] = {X 364.4852, Y 65.5842, Z -1.3333, A 0.000, B 0.000, C 0.000 }
gfCNCPoint1[1569] = {X 363.5690, Y 64.4564, Z -1.3333, A 0.000, B 0.000, C 0.000 }
gfCNCPoint1[1570] = {X 362.8320, Y 63.2041, Z -1.3333, A 0.000, B 0.000, C 0.000 }
gfCNCPoint1[1571] = {X 362.2907, Y 61.8556, Z -1.3333, A 0.000, B 0.000, C 0.000 }
gfCNCPoint1[1572] = {X 361.9573, Y 60.4413, Z -1.3333, A 0.000, B 0.000, C 0.000 }
gfCNCPoint1[1573] = {X 361.8395, Y 58.9930, Z -1.3333, A 0.000, B 0.000, C 0.000 }
gfCNCPoint1[1574] = {X 361.8393, Y 58.0000, Z -1.3333, A 0.000, B 0.000, C 0.000 }
gfCNCPoint1[1575] = {X 361.9156, Y 56.7868, Z -1.3333, A 0.000, B 0.000, C 0.000 }
gfCNCPoint1[1576] = {X 362.1434, Y 55.5928, Z -1.3333, A 0.000, B 0.000, C 0.000 }
gfCNCPoint1[1577] = {X 362.5748, Y 54.2987, Z -1.3333, A 0.000, B 0.000, C 0.000 }
gfCNCPoint1[1578] = {X 363.1839, Y 53.0782, Z -1.3333, A 0.000, B 0.000, C 0.000 }
gfCNCPoint1[1579] = {X 363.9585, Y 51.9554, Z -1.3333, A 0.000, B 0.000, C 0.000 }
gfCNCPoint1[1580] = {X 364.8833, Y 50.9526, Z -1.3333, A 0.000, B 0.000, C 0.000 }
gfCNCPoint1[1581] = {X 365.9398, Y 50.0898, Z -1.3333, A 0.000, B 0.000, C 0.000 }
gfCNCPoint1[1582] = {X 367.1071, Y 49.3840, Z -1.3333, A 0.000, B 0.000, C 0.000 }
gfCNCPoint1[1583] = {X 368.3621, Y 48.8494, Z -1.3333, A 0.000, B 0.000, C 0.000 }
gfCNCPoint1[1584] = {X 369.6797, Y 48.4964, Z -1.3333, A 0.000, B 0.000, C 0.000 }
gfCNCPoint1[1585] = {X 371.0339, Y 48.3322, Z -1.3333, A 0.000, B 0.000, C 0.000 }
gfCNCPoint1[1586] = {X 371.2765, Y 48.3230, Z -1.3333, A 0.000, B 0.000, C 0.000 }
gfCNCPoint1[1587] = {X 371.5193, Y 48.3200, Z -1.3333, A 0.000, B 0.000, C 0.000 }
gfCNCPoint1[1588] = {X 388.0597, Y 48.3200, Z -1.3333, A 0.000, B 0.000, C 0.000 }
gfCNCPoint1[1589] = {X 389.4419, Y 48.4192, Z -1.3333, A 0.000, B 0.000, C 0.000 }
gfCNCPoint1[1590] = {X 390.7958, Y 48.7147, Z -1.3333, A 0.000, B 0.000, C 0.000 }
gfCNCPoint1[1591] = {X 392.0936, Y 49.2006, Z -1.3333, A 0.000, B 0.000, C 0.000 }
gfCNCPoint1[1592] = {X 393.3087, Y 49.8667, Z -1.3333, A 0.000, B 0.000, C 0.000 }
gfCNCPoint1[1593] = {X 394.5333, Y 49.1962, Z -1.3333, A 0.000, B 0.000, C 0.000 }
gfCNCPoint1[1594] = {X 395.8416, Y 48.7089, Z -1.3333, A 0.000, B 0.000, C 0.000 }
gfCNCPoint1[1595] = {X 397.1858, Y 48.4177, Z -1.3333, A 0.000, B 0.000, C 0.000 }
gfCNCPoint1[1596] = {X 398.5577, Y 48.3200, Z -1.3333, A 0.000, B 0.000, C 0.000 }
gfCNCPoint1[1597] = {X 398.7346, Y 48.3200, Z -1.3333, A 0.000, B 0.000, C 0.000 }
gfCNCPoint1[1598] = {X 398.1859, Y 47.6069, Z -1.3333, A 0.000, B 0.000, C 0.000 }
gfCNCPoint1[1599] = {X 397.7774, Y 46.8051, Z -1.3333, A 0.000, B 0.000, C 0.000 }
gfCNCPoint1[1600] = {X 397.5230, Y 45.9420, Z -1.3333, A 0.000, B 0.000, C 0.000 }
gfCNCPoint1[1601] = {X 397.4561, Y 45.4921, Z -1.3333, A 0.000, B 0.000, C 0.000 }
gfCNCPoint1[1602] = {X 397.4314, Y 45.0378, Z -1.3333, A 0.000, B 0.000, C 0.000 }
gfCNCPoint1[1603] = {X 397.4316, Y 44.1456, Z -1.3333, A 0.000, B 0.000, C 0.000 }
gfCNCPoint1[1604] = {X 397.5413, Y 43.1780, Z -1.3333, A 0.000, B 0.000, C 0.000 }
gfCNCPoint1[1605] = {X 397.8410, Y 42.2514, Z -1.3333, A 0.000, B 0.000, C 0.000 }
gfCNCPoint1[1606] = {X 398.3186, Y 41.4029, Z -1.3333, A 0.000, B 0.000, C 0.000 }
gfCNCPoint1[1607] = {X 398.9552, Y 40.6660, Z -1.3333, A 0.000, B 0.000, C 0.000 }
gfCNCPoint1[1608] = {X 398.9552, Y 31.8209, Z -1.3333, A 0.000, B 0.000, C 0.000 }
gfCNCPoint1[1609] = {X 396.7494, Y 27.9853, Z -1.3333, A 0.000, B 0.000, C 0.000 }
gfCNCPoint1[1610] = {X 386.3469, Y 33.9675, Z -1.3333, A 0.000, B 0.000, C 0.000 }
gfCNCPoint1[1611] = {X 386.2659, Y 34.3953, Z -1.3333, A 0.000, B 0.000, C 0.000 }
gfCNCPoint1[1612] = {X 386.1812, Y 34.8223, Z -1.3333, A 0.000, B 0.000, C 0.000 }
gfCNCPoint1[1613] = {X 386.0220, Y 35.5727, Z -1.3333, A 0.000, B 0.000, C 0.000 }
gfCNCPoint1[1614] = {X 385.8491, Y 36.3200, Z -1.3333, A 0.000, B 0.000, C 0.000 }
gfCNCPoint1[1615] = {X 386.9552, Y 36.3200, Z -1.3333, A 0.000, B 0.000, C 0.000 }
gfCNCPoint1[1616] = {X 386.9552, Y 35.0253, Z -1.3333, A 0.000, B 0.000, C 0.000 }
gfCNCPoint1[1617] = {X 386.3469, Y 33.9675, Z -1.3333, A 0.000, B 0.000, C 0.000 }
gfCNCPoint1[1618] = {X 388.4274, Y 32.7711, Z -1.3333, A 0.000, B 0.000, C 0.000 }
gfCNCPoint1[1619] = {X 384.7435, Y 26.3652, Z -1.3333, A 0.000, B 0.000, C 0.000 }
gfCNCPoint1[1620] = {X 384.6147, Y 28.7660, Z -1.3333, A 0.000, B 0.000, C 0.000 }
gfCNCPoint1[1621] = {X 384.3622, Y 31.1569, Z -1.3333, A 0.000, B 0.000, C 0.000 }
gfCNCPoint1[1622] = {X 383.9868, Y 33.5317, Z -1.3333, A 0.000, B 0.000, C 0.000 }
gfCNCPoint1[1623] = {X 383.9097, Y 33.9388, Z -1.3333, A 0.000, B 0.000, C 0.000 }
gfCNCPoint1[1624] = {X 383.8291, Y 34.3452, Z -1.3333, A 0.000, B 0.000, C 0.000 }
gfCNCPoint1[1625] = {X 383.6790, Y 35.0529, Z -1.3333, A 0.000, B 0.000, C 0.000 }
gfCNCPoint1[1626] = {X 383.5159, Y 35.7577, Z -1.3333, A 0.000, B 0.000, C 0.000 }
gfCNCPoint1[1627] = {X 383.1261, Y 37.2470, Z -1.3333, A 0.000, B 0.000, C 0.000 }
gfCNCPoint1[1628] = {X 382.6785, Y 38.7200, Z -1.3333, A 0.000, B 0.000, C 0.000 }
gfCNCPoint1[1629] = {X 388.0597, Y 38.7200, Z -1.3333, A 0.000, B 0.000, C 0.000 }
gfCNCPoint1[1630] = {X 388.4821, Y 38.7246, Z -1.3333, A 0.000, B 0.000, C 0.000 }
gfCNCPoint1[1631] = {X 388.9043, Y 38.7385, Z -1.3333, A 0.000, B 0.000, C 0.000 }
gfCNCPoint1[1632] = {X 389.1204, Y 38.2363, Z -1.3333, A 0.000, B 0.000, C 0.000 }
gfCNCPoint1[1633] = {X 389.3552, Y 37.7427, Z -1.3333, A 0.000, B 0.000, C 0.000 }
gfCNCPoint1[1634] = {X 389.3552, Y 34.3844, Z -1.3333, A 0.000, B 0.000, C 0.000 }
gfCNCPoint1[1635] = {X 388.4274, Y 32.7711, Z -1.3333, A 0.000, B 0.000, C 0.000 }
gfCNCPoint1[1636] = {X 390.5079, Y 31.5746, Z -1.3333, A 0.000, B 0.000, C 0.000 }
gfCNCPoint1[1637] = {X 386.6280, Y 24.8278, Z -1.3333, A 0.000, B 0.000, C 0.000 }
gfCNCPoint1[1638] = {X 386.0726, Y 23.8807, Z -1.3333, A 0.000, B 0.000, C 0.000 }
gfCNCPoint1[1639] = {X 385.5014, Y 22.9430, Z -1.3333, A 0.000, B 0.000, C 0.000 }
gfCNCPoint1[1640] = {X 384.4715, Y 22.1528, Z -1.3333, A 0.000, B 0.000, C 0.000 }
gfCNCPoint1[1641] = {X 383.5324, Y 21.2566, Z -1.3333, A 0.000, B 0.000, C 0.000 }
gfCNCPoint1[1642] = {X 382.6948, Y 20.2648, Z -1.3333, A 0.000, B 0.000, C 0.000 }
gfCNCPoint1[1643] = {X 381.9685, Y 19.1888, Z -1.3333, A 0.000, B 0.000, C 0.000 }
gfCNCPoint1[1644] = {X 382.2212, Y 21.5508, Z -1.3333, A 0.000, B 0.000, C 0.000 }
gfCNCPoint1[1645] = {X 382.3466, Y 23.9230, Z -1.3333, A 0.000, B 0.000, C 0.000 }
gfCNCPoint1[1646] = {X 382.3444, Y 26.2985, Z -1.3333, A 0.000, B 0.000, C 0.000 }
gfCNCPoint1[1647] = {X 382.2007, Y 28.8369, Z -1.3333, A 0.000, B 0.000, C 0.000 }
gfCNCPoint1[1648] = {X 381.9112, Y 31.3630, Z -1.3333, A 0.000, B 0.000, C 0.000 }
gfCNCPoint1[1649] = {X 381.4770, Y 33.8682, Z -1.3333, A 0.000, B 0.000, C 0.000 }
gfCNCPoint1[1650] = {X 380.9955, Y 35.9383, Z -1.3333, A 0.000, B 0.000, C 0.000 }
gfCNCPoint1[1651] = {X 380.3962, Y 37.9775, Z -1.3333, A 0.000, B 0.000, C 0.000 }
gfCNCPoint1[1652] = {X 379.8407, Y 39.5622, Z -1.3333, A 0.000, B 0.000, C 0.000 }
gfCNCPoint1[1653] = {X 379.2140, Y 41.1200, Z -1.3333, A 0.000, B 0.000, C 0.000 }
gfCNCPoint1[1654] = {X 388.0597, Y 41.1200, Z -1.3333, A 0.000, B 0.000, C 0.000 }
gfCNCPoint1[1655] = {X 389.3256, Y 41.1675, Z -1.3333, A 0.000, B 0.000, C 0.000 }
gfCNCPoint1[1656] = {X 390.5843, Y 41.3099, Z -1.3333, A 0.000, B 0.000, C 0.000 }
gfCNCPoint1[1657] = {X 391.0709, Y 39.7838, Z -1.3333, A 0.000, B 0.000, C 0.000 }
gfCNCPoint1[1658] = {X 391.7552, Y 38.3355, Z -1.3333, A 0.000, B 0.000, C 0.000 }
gfCNCPoint1[1659] = {X 391.7552, Y 33.7435, Z -1.3333, A 0.000, B 0.000, C 0.000 }
gfCNCPoint1[1660] = {X 390.5079, Y 31.5746, Z -1.3333, A 0.000, B 0.000, C 0.000 }
gfCNCPoint1[1661] = {X 392.5884, Y 30.3782, Z -1.3333, A 0.000, B 0.000, C 0.000 }
gfCNCPoint1[1662] = {X 388.7085, Y 23.6314, Z -1.3333, A 0.000, B 0.000, C 0.000 }
gfCNCPoint1[1663] = {X 387.9941, Y 22.4186, Z -1.3333, A 0.000, B 0.000, C 0.000 }
gfCNCPoint1[1664] = {X 387.2547, Y 21.2210, Z -1.3333, A 0.000, B 0.000, C 0.000 }
gfCNCPoint1[1665] = {X 386.3064, Y 20.5558, Z -1.3333, A 0.000, B 0.000, C 0.000 }
gfCNCPoint1[1666] = {X 385.4444, Y 19.7821, Z -1.3333, A 0.000, B 0.000, C 0.000 }
gfCNCPoint1[1667] = {X 384.6809, Y 18.9110, Z -1.3333, A 0.000, B 0.000, C 0.000 }
gfCNCPoint1[1668] = {X 384.0270, Y 17.9549, Z -1.3333, A 0.000, B 0.000, C 0.000 }
gfCNCPoint1[1669] = {X 383.4393, Y 16.8074, Z -1.3333, A 0.000, B 0.000, C 0.000 }
gfCNCPoint1[1670] = {X 383.0092, Y 15.5919, Z -1.3333, A 0.000, B 0.000, C 0.000 }
gfCNCPoint1[1671] = {X 382.7445, Y 14.3301, Z -1.3333, A 0.000, B 0.000, C 0.000 }
gfCNCPoint1[1672] = {X 382.6498, Y 13.0443, Z -1.3333, A 0.000, B 0.000, C 0.000 }
gfCNCPoint1[1673] = {X 382.6496, Y 12.1868, Z -1.3333, A 0.000, B 0.000, C 0.000 }
gfCNCPoint1[1674] = {X 382.6507, Y 12.0459, Z -1.3333, A 0.000, B 0.000, C 0.000 }
gfCNCPoint1[1675] = {X 382.6537, Y 11.9051, Z -1.3333, A 0.000, B 0.000, C 0.000 }
gfCNCPoint1[1676] = {X 377.7920, Y 11.9051, Z -1.3333, A 0.000, B 0.000, C 0.000 }
gfCNCPoint1[1677] = {X 378.4211, Y 13.8642, Z -1.3333, A 0.000, B 0.000, C 0.000 }
gfCNCPoint1[1678] = {X 378.9336, Y 15.8570, Z -1.3333, A 0.000, B 0.000, C 0.000 }
gfCNCPoint1[1679] = {X 379.3023, Y 17.6753, Z -1.3333, A 0.000, B 0.000, C 0.000 }
gfCNCPoint1[1680] = {X 379.5899, Y 19.5082, Z -1.3333, A 0.000, B 0.000, C 0.000 }
gfCNCPoint1[1681] = {X 379.8686, Y 22.2848, Z -1.3333, A 0.000, B 0.000, C 0.000 }
gfCNCPoint1[1682] = {X 379.9615, Y 25.0738, Z -1.3333, A 0.000, B 0.000, C 0.000 }
gfCNCPoint1[1683] = {X 379.8681, Y 27.8628, Z -1.3333, A 0.000, B 0.000, C 0.000 }
gfCNCPoint1[1684] = {X 379.5888, Y 30.6393, Z -1.3333, A 0.000, B 0.000, C 0.000 }
gfCNCPoint1[1685] = {X 379.1249, Y 33.3911, Z -1.3333, A 0.000, B 0.000, C 0.000 }
gfCNCPoint1[1686] = {X 378.5747, Y 35.6986, Z -1.3333, A 0.000, B 0.000, C 0.000 }
gfCNCPoint1[1687] = {X 377.8681, Y 37.9632, Z -1.3333, A 0.000, B 0.000, C 0.000 }
gfCNCPoint1[1688] = {X 377.0083, Y 40.1741, Z -1.3333, A 0.000, B 0.000, C 0.000 }
gfCNCPoint1[1689] = {X 376.2266, Y 41.8693, Z -1.3333, A 0.000, B 0.000, C 0.000 }
gfCNCPoint1[1690] = {X 375.3549, Y 43.5200, Z -1.3333, A 0.000, B 0.000, C 0.000 }
gfCNCPoint1[1691] = {X 388.0597, Y 43.5200, Z -1.3333, A 0.000, B 0.000, C 0.000 }
gfCNCPoint1[1692] = {X 389.6072, Y 43.6029, Z -1.3333, A 0.000, B 0.000, C 0.000 }
gfCNCPoint1[1693] = {X 391.1370, Y 43.8508, Z -1.3333, A 0.000, B 0.000, C 0.000 }
gfCNCPoint1[1694] = {X 392.6316, Y 44.2607, Z -1.3333, A 0.000, B 0.000, C 0.000 }
gfCNCPoint1[1695] = {X 392.7236, Y 42.8756, Z -1.3333, A 0.000, B 0.000, C 0.000 }
gfCNCPoint1[1696] = {X 393.0129, Y 41.5179, Z -1.3333, A 0.000, B 0.000, C 0.000 }
gfCNCPoint1[1697] = {X 393.4934, Y 40.2155, Z -1.3333, A 0.000, B 0.000, C 0.000 }
gfCNCPoint1[1698] = {X 394.1552, Y 38.9952, Z -1.3333, A 0.000, B 0.000, C 0.000 }
gfCNCPoint1[1699] = {X 394.1552, Y 33.1027, Z -1.3333, A 0.000, B 0.000, C 0.000 }
gfCNCPoint1[1700] = {X 392.5884, Y 30.3782, Z -1.3333, A 0.000, B 0.000, C 0.000 }
gfCNCPoint1[1701] = {X 394.6689, Y 29.1817, Z -1.3333, A 0.000, B 0.000, C 0.000 }
gfCNCPoint1[1702] = {X 390.7890, Y 22.4349, Z -1.3333, A 0.000, B 0.000, C 0.000 }
gfCNCPoint1[1703] = {X 389.9897, Y 21.0805, Z -1.3333, A 0.000, B 0.000, C 0.000 }
gfCNCPoint1[1704] = {X 389.1601, Y 19.7444, Z -1.3333, A 0.000, B 0.000, C 0.000 }
gfCNCPoint1[1705] = {X 389.0413, Y 19.5708, Z -1.3333, A 0.000, B 0.000, C 0.000 }
gfCNCPoint1[1706] = {X 388.9111, Y 19.4054, Z -1.3333, A 0.000, B 0.000, C 0.000 }
gfCNCPoint1[1707] = {X 387.8211, Y 18.6939, Z -1.3333, A 0.000, B 0.000, C 0.000 }
gfCNCPoint1[1708] = {X 386.8753, Y 17.7997, Z -1.3333, A 0.000, B 0.000, C 0.000 }
gfCNCPoint1[1709] = {X 386.1038, Y 16.7513, Z -1.3333, A 0.000, B 0.000, C 0.000 }
gfCNCPoint1[1710] = {X 385.5314, Y 15.5824, Z -1.3333, A 0.000, B 0.000, C 0.000 }
gfCNCPoint1[1711] = {X 385.1763, Y 14.3301, Z -1.3333, A 0.000, B 0.000, C 0.000 }
gfCNCPoint1[1712] = {X 385.0498, Y 13.0347, Z -1.3333, A 0.000, B 0.000, C 0.000 }
gfCNCPoint1[1713] = {X 385.0496, Y 12.1868, Z -1.3333, A 0.000, B 0.000, C 0.000 }
gfCNCPoint1[1714] = {X 385.0504, Y 12.0809, Z -1.3333, A 0.000, B 0.000, C 0.000 }
gfCNCPoint1[1715] = {X 385.0527, Y 11.9750, Z -1.3333, A 0.000, B 0.000, C 0.000 }
gfCNCPoint1[1716] = {X 385.1994, Y 10.7178, Z -1.3333, A 0.000, B 0.000, C 0.000 }
gfCNCPoint1[1717] = {X 385.5616, Y 9.5051, Z -1.3333, A 0.000, B 0.000, C 0.000 }
gfCNCPoint1[1718] = {X 374.2003, Y 9.5051, Z -1.3333, A 0.000, B 0.000, C 0.000 }
gfCNCPoint1[1719] = {X 374.9076, Y 11.0878, Z -1.3333, A 0.000, B 0.000, C 0.000 }
gfCNCPoint1[1720] = {X 375.5295, Y 12.7060, Z -1.3333, A 0.000, B 0.000, C 0.000 }
gfCNCPoint1[1721] = {X 376.1154, Y 14.5303, Z -1.3333, A 0.000, B 0.000, C 0.000 }
gfCNCPoint1[1722] = {X 376.5926, Y 16.3860, Z -1.3333, A 0.000, B 0.000, C 0.000 }
gfCNCPoint1[1723] = {X 377.1085, Y 19.1125, Z -1.3333, A 0.000, B 0.000, C 0.000 }
gfCNCPoint1[1724] = {X 377.4313, Y 21.8685, Z -1.3333, A 0.000, B 0.000, C 0.000 }
gfCNCPoint1[1725] = {X 377.5592, Y 24.6404, Z -1.3333, A 0.000, B 0.000, C 0.000 }
gfCNCPoint1[1726] = {X 377.4917, Y 27.4145, Z -1.3333, A 0.000, B 0.000, C 0.000 }
gfCNCPoint1[1727] = {X 377.2291, Y 30.1769, Z -1.3333, A 0.000, B 0.000, C 0.000 }
gfCNCPoint1[1728] = {X 376.7728, Y 32.9140, Z -1.3333, A 0.000, B 0.000, C 0.000 }
gfCNCPoint1[1729] = {X 376.1753, Y 35.3670, Z -1.3333, A 0.000, B 0.000, C 0.000 }
gfCNCPoint1[1730] = {X 375.3878, Y 37.7658, Z -1.3333, A 0.000, B 0.000, C 0.000 }
gfCNCPoint1[1731] = {X 374.4153, Y 40.0957, Z -1.3333, A 0.000, B 0.000, C 0.000 }
gfCNCPoint1[1732] = {X 373.2636, Y 42.3425, Z -1.3333, A 0.000, B 0.000, C 0.000 }
gfCNCPoint1[1733] = {X 372.1856, Y 44.1205, Z -1.3333, A 0.000, B 0.000, C 0.000 }
gfCNCPoint1[1734] = {X 370.9954, Y 45.8254, Z -1.3333, A 0.000, B 0.000, C 0.000 }
gfCNCPoint1[1735] = {X 370.9135, Y 45.9352, Z -1.3333, A 0.000, B 0.000, C 0.000 }
gfCNCPoint1[1736] = {X 371.2163, Y 45.9238, Z -1.3333, A 0.000, B 0.000, C 0.000 }
gfCNCPoint1[1737] = {X 371.5193, Y 45.9200, Z -1.3333, A 0.000, B 0.000, C 0.000 }
gfCNCPoint1[1738] = {X 388.0597, Y 45.9200, Z -1.3333, A 0.000, B 0.000, C 0.000 }
gfCNCPoint1[1739] = {X 389.4143, Y 45.9962, Z -1.3333, A 0.000, B 0.000, C 0.000 }
gfCNCPoint1[1740] = {X 390.7519, Y 46.2238, Z -1.3333, A 0.000, B 0.000, C 0.000 }
gfCNCPoint1[1741] = {X 392.0555, Y 46.6000, Z -1.3333, A 0.000, B 0.000, C 0.000 }
gfCNCPoint1[1742] = {X 393.3087, Y 47.1200, Z -1.3333, A 0.000, B 0.000, C 0.000 }
gfCNCPoint1[1743] = {X 394.2237, Y 46.7243, Z -1.3333, A 0.000, B 0.000, C 0.000 }
gfCNCPoint1[1744] = {X 395.1681, Y 46.4053, Z -1.3333, A 0.000, B 0.000, C 0.000 }
gfCNCPoint1[1745] = {X 395.0678, Y 45.7292, Z -1.3333, A 0.000, B 0.000, C 0.000 }
gfCNCPoint1[1746] = {X 395.0314, Y 45.0468, Z -1.3333, A 0.000, B 0.000, C 0.000 }
gfCNCPoint1[1747] = {X 395.0316, Y 44.1297, Z -1.3333, A 0.000, B 0.000, C 0.000 }
gfCNCPoint1[1748] = {X 395.1397, Y 42.9565, Z -1.3333, A 0.000, B 0.000, C 0.000 }
gfCNCPoint1[1749] = {X 395.4356, Y 41.8161, Z -1.3333, A 0.000, B 0.000, C 0.000 }
gfCNCPoint1[1750] = {X 395.9116, Y 40.7384, Z -1.3333, A 0.000, B 0.000, C 0.000 }
gfCNCPoint1[1751] = {X 396.5552, Y 39.7516, Z -1.3333, A 0.000, B 0.000, C 0.000 }
gfCNCPoint1[1752] = {X 396.5552, Y 32.4618, Z -1.3333, A 0.000, B 0.000, C 0.000 }
gfCNCPoint1[1753] = {X 394.6689, Y 29.1817, Z -1.3333, A 0.000, B 0.000, C 0.000 }
gfCNCPoint1[1754] = {X 396.7494, Y 27.9853, Z -1.3333, A 0.000, B 0.000, C 0.000 }
gfCNCPoint1[1755] = {X 392.8695, Y 21.2385, Z -1.3333, A 0.000, B 0.000, C 0.000 }
gfCNCPoint1[1756] = {X 392.0428, Y 19.8376, Z -1.3333, A 0.000, B 0.000, C 0.000 }
gfCNCPoint1[1757] = {X 391.1847, Y 18.4556, Z -1.3333, A 0.000, B 0.000, C 0.000 }
gfCNCPoint1[1758] = {X 390.8000, Y 17.9236, Z -1.3333, A 0.000, B 0.000, C 0.000 }
gfCNCPoint1[1759] = {X 390.3552, Y 17.4408, Z -1.3333, A 0.000, B 0.000, C 0.000 }
gfCNCPoint1[1760] = {X 389.5446, Y 16.9853, Z -1.3333, A 0.000, B 0.000, C 0.000 }
gfCNCPoint1[1761] = {X 388.8351, Y 16.3842, Z -1.3333, A 0.000, B 0.000, C 0.000 }
gfCNCPoint1[1762] = {X 388.2524, Y 15.6596, Z -1.3333, A 0.000, B 0.000, C 0.000 }
gfCNCPoint1[1763] = {X 387.8178, Y 14.8375, Z -1.3333, A 0.000, B 0.000, C 0.000 }
gfCNCPoint1[1764] = {X 387.5470, Y 13.9480, Z -1.3333, A 0.000, B 0.000, C 0.000 }
gfCNCPoint1[1765] = {X 387.4498, Y 13.0232, Z -1.3333, A 0.000, B 0.000, C 0.000 }
gfCNCPoint1[1766] = {X 387.4496, Y 12.1868, Z -1.3333, A 0.000, B 0.000, C 0.000 }
gfCNCPoint1[1767] = {X 387.5362, Y 11.2718, Z -1.3333, A 0.000, B 0.000, C 0.000 }
gfCNCPoint1[1768] = {X 387.7928, Y 10.3892, Z -1.3333, A 0.000, B 0.000, C 0.000 }
gfCNCPoint1[1769] = {X 388.2375, Y 9.5281, Z -1.3333, A 0.000, B 0.000, C 0.000 }
gfCNCPoint1[1770] = {X 388.8436, Y 8.7719, Z -1.3333, A 0.000, B 0.000, C 0.000 }
gfCNCPoint1[1771] = {X 389.5872, Y 8.1503, Z -1.3333, A 0.000, B 0.000, C 0.000 }
gfCNCPoint1[1772] = {X 390.4389, Y 7.6880, Z -1.3333, A 0.000, B 0.000, C 0.000 }
gfCNCPoint1[1773] = {X 391.3653, Y 7.4030, Z -1.3333, A 0.000, B 0.000, C 0.000 }
gfCNCPoint1[1774] = {X 392.3296, Y 7.3068, Z -1.3333, A 0.000, B 0.000, C 0.000 }
gfCNCPoint1[1775] = {X 399.1118, Y 7.3068, Z -1.3333, A 0.000, B 0.000, C 0.000 }
gfCNCPoint1[1776] = {X 400.0638, Y 7.4006, Z -1.3333, A 0.000, B 0.000, C 0.000 }
gfCNCPoint1[1777] = {X 400.9793, Y 7.6783, Z -1.3333, A 0.000, B 0.000, C 0.000 }
gfCNCPoint1[1778] = {X 401.8229, Y 8.1292, Z -1.3333, A 0.000, B 0.000, C 0.000 }
gfCNCPoint1[1779] = {X 402.5624, Y 8.7361, Z -1.3333, A 0.000, B 0.000, C 0.000 }
gfCNCPoint1[1780] = {X 403.1693, Y 9.4756, Z -1.3333, A 0.000, B 0.000, C 0.000 }
gfCNCPoint1[1781] = {X 403.6203, Y 10.3193, Z -1.3333, A 0.000, B 0.000, C 0.000 }
gfCNCPoint1[1782] = {X 403.8980, Y 11.2348, Z -1.3333, A 0.000, B 0.000, C 0.000 }
gfCNCPoint1[1783] = {X 403.9918, Y 12.1868, Z -1.3333, A 0.000, B 0.000, C 0.000 }
gfCNCPoint1[1784] = {X 403.9915, Y 13.0237, Z -1.3333, A 0.000, B 0.000, C 0.000 }
gfCNCPoint1[1785] = {X 403.9016, Y 13.9115, Z -1.3333, A 0.000, B 0.000, C 0.000 }
gfCNCPoint1[1786] = {X 403.6516, Y 14.7680, Z -1.3333, A 0.000, B 0.000, C 0.000 }
gfCNCPoint1[1787] = {X 405.3655, Y 17.7440, Z -1.3333, A 0.000, B 0.000, C 0.000 }
gfCNCPoint1[1788] = {X 407.2451, Y 14.6992, Z -1.3333, A 0.000, B 0.000, C 0.000 }
gfCNCPoint1[1789] = {X 407.0144, Y 13.8734, Z -1.3333, A 0.000, B 0.000, C 0.000 }
gfCNCPoint1[1790] = {X 406.9317, Y 13.0199, Z -1.3333, A 0.000, B 0.000, C 0.000 }
gfCNCPoint1[1791] = {X 406.9315, Y 12.1868, Z -1.3333, A 0.000, B 0.000, C 0.000 }
gfCNCPoint1[1792] = {X 407.0253, Y 11.2348, Z -1.3333, A 0.000, B 0.000, C 0.000 }
gfCNCPoint1[1793] = {X 407.3030, Y 10.3193, Z -1.3333, A 0.000, B 0.000, C 0.000 }
gfCNCPoint1[1794] = {X 407.7540, Y 9.4756, Z -1.3333, A 0.000, B 0.000, C 0.000 }
gfCNCPoint1[1795] = {X 408.3609, Y 8.7361, Z -1.3333, A 0.000, B 0.000, C 0.000 }
gfCNCPoint1[1796] = {X 409.1004, Y 8.1292, Z -1.3333, A 0.000, B 0.000, C 0.000 }
gfCNCPoint1[1797] = {X 409.9440, Y 7.6783, Z -1.3333, A 0.000, B 0.000, C 0.000 }
gfCNCPoint1[1798] = {X 410.8595, Y 7.4006, Z -1.3333, A 0.000, B 0.000, C 0.000 }
gfCNCPoint1[1799] = {X 411.8115, Y 7.3068, Z -1.3333, A 0.000, B 0.000, C 0.000 }
gfCNCPoint1[1800] = {X 419.3245, Y 7.3068, Z -1.3333, A 0.000, B 0.000, C 0.000 }
gfCNCPoint1[1801] = {X 420.2888, Y 7.4030, Z -1.3333, A 0.000, B 0.000, C 0.000 }
gfCNCPoint1[1802] = {X 421.2151, Y 7.6880, Z -1.3333, A 0.000, B 0.000, C 0.000 }
gfCNCPoint1[1803] = {X 422.0669, Y 8.1503, Z -1.3333, A 0.000, B 0.000, C 0.000 }
gfCNCPoint1[1804] = {X 422.8105, Y 8.7719, Z -1.3333, A 0.000, B 0.000, C 0.000 }
gfCNCPoint1[1805] = {X 423.4166, Y 9.5281, Z -1.3333, A 0.000, B 0.000, C 0.000 }
gfCNCPoint1[1806] = {X 423.8613, Y 10.3892, Z -1.3333, A 0.000, B 0.000, C 0.000 }
gfCNCPoint1[1807] = {X 424.1179, Y 11.2718, Z -1.3333, A 0.000, B 0.000, C 0.000 }
gfCNCPoint1[1808] = {X 424.2045, Y 12.1868, Z -1.3333, A 0.000, B 0.000, C 0.000 }
gfCNCPoint1[1809] = {X 424.2045, Y 12.9779, Z -1.3333, A 0.000, B 0.000, C 0.000 }
gfCNCPoint1[1810] = {X 424.1054, Y 13.9306, Z -1.3333, A 0.000, B 0.000, C 0.000 }
gfCNCPoint1[1811] = {X 423.8246, Y 14.8464, Z -1.3333, A 0.000, B 0.000, C 0.000 }
gfCNCPoint1[1812] = {X 423.3726, Y 15.6909, Z -1.3333, A 0.000, B 0.000, C 0.000 }
gfCNCPoint1[1813] = {X 422.7664, Y 16.4326, Z -1.3333, A 0.000, B 0.000, C 0.000 }
gfCNCPoint1[1814] = {X 422.0287, Y 17.0435, Z -1.3333, A 0.000, B 0.000, C 0.000 }
gfCNCPoint1[1815] = {X 421.1871, Y 17.5008, Z -1.3333, A 0.000, B 0.000, C 0.000 }
gfCNCPoint1[1816] = {X 420.5393, Y 18.3844, Z -1.3333, A 0.000, B 0.000, C 0.000 }
gfCNCPoint1[1817] = {X 419.9500, Y 19.3080, Z -1.3333, A 0.000, B 0.000, C 0.000 }
gfCNCPoint1[1818] = {X 414.1631, Y 28.6156, Z -1.3333, A 0.000, B 0.000, C 0.000 }
gfCNCPoint1[1819] = {X 422.3159, Y 33.6844, Z -1.3333, A 0.000, B 0.000, C 0.000 }
gfCNCPoint1[1820] = {X 421.8880, Y 34.3727, Z -1.3333, A 0.000, B 0.000, C 0.000 }
gfCNCPoint1[1821] = {X 422.1452, Y 34.1019, Z -1.3333, A 0.000, B 0.000, C 0.000 }
gfCNCPoint1[1822] = {X 422.4093, Y 33.8378, Z -1.3333, A 0.000, B 0.000, C 0.000 }
gfCNCPoint1[1823] = {X 422.3624, Y 33.7612, Z -1.3333, A 0.000, B 0.000, C 0.000 }
gfCNCPoint1[1824] = {X 422.3159, Y 33.6844, Z -1.3333, A 0.000, B 0.000, C 0.000 }
gfCNCPoint1[1825] = {X 420.2777, Y 32.4172, Z -1.3333, A 0.000, B 0.000, C 0.000 }
gfCNCPoint1[1826] = {X 419.3058, Y 33.9804, Z -1.3333, A 0.000, B 0.000, C 0.000 }
gfCNCPoint1[1827] = {X 419.3062, Y 38.3390, Z -1.3333, A 0.000, B 0.000, C 0.000 }
gfCNCPoint1[1828] = {X 419.9568, Y 39.7077, Z -1.3333, A 0.000, B 0.000, C 0.000 }
gfCNCPoint1[1829] = {X 420.4328, Y 41.1464, Z -1.3333, A 0.000, B 0.000, C 0.000 }
gfCNCPoint1[1830] = {X 420.6275, Y 41.1585, Z -1.3333, A 0.000, B 0.000, C 0.000 }
gfCNCPoint1[1831] = {X 420.8221, Y 41.1728, Z -1.3333, A 0.000, B 0.000, C 0.000 }
gfCNCPoint1[1832] = {X 421.2838, Y 39.7591, Z -1.3333, A 0.000, B 0.000, C 0.000 }
gfCNCPoint1[1833] = {X 421.9157, Y 38.4129, Z -1.3333, A 0.000, B 0.000, C 0.000 }
gfCNCPoint1[1834] = {X 422.7081, Y 37.1545, Z -1.3333, A 0.000, B 0.000, C 0.000 }
gfCNCPoint1[1835] = {X 423.6492, Y 36.0030, Z -1.3333, A 0.000, B 0.000, C 0.000 }
gfCNCPoint1[1836] = {X 424.3395, Y 35.3152, Z -1.3333, A 0.000, B 0.000, C 0.000 }
gfCNCPoint1[1837] = {X 425.0829, Y 34.6852, Z -1.3333, A 0.000, B 0.000, C 0.000 }
gfCNCPoint1[1838] = {X 425.4265, Y 34.0126, Z -1.3333, A 0.000, B 0.000, C 0.000 }
gfCNCPoint1[1839] = {X 424.8791, Y 33.2415, Z -1.3333, A 0.000, B 0.000, C 0.000 }
gfCNCPoint1[1840] = {X 424.3707, Y 32.4443, Z -1.3333, A 0.000, B 0.000, C 0.000 }
gfCNCPoint1[1841] = {X 423.3899, Y 30.5975, Z -1.3333, A 0.000, B 0.000, C 0.000 }
gfCNCPoint1[1842] = {X 422.6171, Y 28.6544, Z -1.3333, A 0.000, B 0.000, C 0.000 }
gfCNCPoint1[1843] = {X 420.2777, Y 32.4172, Z -1.3333, A 0.000, B 0.000, C 0.000 }
gfCNCPoint1[1844] = {X 418.2395, Y 31.1500, Z -1.3333, A 0.000, B 0.000, C 0.000 }
gfCNCPoint1[1845] = {X 416.9058, Y 33.2952, Z -1.3333, A 0.000, B 0.000, C 0.000 }
gfCNCPoint1[1846] = {X 416.9062, Y 38.9958, Z -1.3333, A 0.000, B 0.000, C 0.000 }
gfCNCPoint1[1847] = {X 417.4877, Y 40.0489, Z -1.3333, A 0.000, B 0.000, C 0.000 }
gfCNCPoint1[1848] = {X 417.9359, Y 41.1653, Z -1.3333, A 0.000, B 0.000, C 0.000 }
gfCNCPoint1[1849] = {X 418.2440, Y 42.3282, Z -1.3333, A 0.000, B 0.000, C 0.000 }
gfCNCPoint1[1850] = {X 418.4074, Y 43.5200, Z -1.3333, A 0.000, B 0.000, C 0.000 }
gfCNCPoint1[1851] = {X 419.4886, Y 43.5200, Z -1.3333, A 0.000, B 0.000, C 0.000 }
gfCNCPoint1[1852] = {X 421.1752, Y 43.6186, Z -1.3333, A 0.000, B 0.000, C 0.000 }
gfCNCPoint1[1853] = {X 422.8389, Y 43.9129, Z -1.3333, A 0.000, B 0.000, C 0.000 }
gfCNCPoint1[1854] = {X 423.0005, Y 42.4234, Z -1.3333, A 0.000, B 0.000, C 0.000 }
gfCNCPoint1[1855] = {X 423.3900, Y 40.9766, Z -1.3333, A 0.000, B 0.000, C 0.000 }
gfCNCPoint1[1856] = {X 423.9980, Y 39.6073, Z -1.3333, A 0.000, B 0.000, C 0.000 }
gfCNCPoint1[1857] = {X 424.8102, Y 38.3482, Z -1.3333, A 0.000, B 0.000, C 0.000 }
gfCNCPoint1[1858] = {X 425.8068, Y 37.2295, Z -1.3333, A 0.000, B 0.000, C 0.000 }
gfCNCPoint1[1859] = {X 426.9642, Y 36.2780, Z -1.3333, A 0.000, B 0.000, C 0.000 }
gfCNCPoint1[1860] = {X 428.2767, Y 33.7089, Z -1.3333, A 0.000, B 0.000, C 0.000 }
gfCNCPoint1[1861] = {X 427.2129, Y 32.3912, Z -1.3333, A 0.000, B 0.000, C 0.000 }
gfCNCPoint1[1862] = {X 426.2881, Y 30.9724, Z -1.3333, A 0.000, B 0.000, C 0.000 }
gfCNCPoint1[1863] = {X 425.5120, Y 29.4672, Z -1.3333, A 0.000, B 0.000, C 0.000 }
gfCNCPoint1[1864] = {X 424.8925, Y 27.8910, Z -1.3333, A 0.000, B 0.000, C 0.000 }
gfCNCPoint1[1865] = {X 424.8108, Y 27.6411, Z -1.3333, A 0.000, B 0.000, C 0.000 }
gfCNCPoint1[1866] = {X 424.7331, Y 27.3899, Z -1.3333, A 0.000, B 0.000, C 0.000 }
gfCNCPoint1[1867] = {X 424.3004, Y 25.6520, Z -1.3333, A 0.000, B 0.000, C 0.000 }
gfCNCPoint1[1868] = {X 424.0108, Y 23.8846, Z -1.3333, A 0.000, B 0.000, C 0.000 }
gfCNCPoint1[1869] = {X 423.8665, Y 22.0995, Z -1.3333, A 0.000, B 0.000, C 0.000 }
gfCNCPoint1[1870] = {X 418.2395, Y 31.1500, Z -1.3333, A 0.000, B 0.000, C 0.000 }
gfCNCPoint1[1871] = {X 416.2013, Y 29.8828, Z -1.3333, A 0.000, B 0.000, C 0.000 }
gfCNCPoint1[1872] = {X 414.5057, Y 32.6100, Z -1.3333, A 0.000, B 0.000, C 0.000 }
gfCNCPoint1[1873] = {X 414.5063, Y 39.7474, Z -1.3333, A 0.000, B 0.000, C 0.000 }
gfCNCPoint1[1874] = {X 415.1549, Y 40.7521, Z -1.3333, A 0.000, B 0.000, C 0.000 }
gfCNCPoint1[1875] = {X 415.6334, Y 41.8482, Z -1.3333, A 0.000, B 0.000, C 0.000 }
gfCNCPoint1[1876] = {X 415.9292, Y 43.0069, Z -1.3333, A 0.000, B 0.000, C 0.000 }
gfCNCPoint1[1877] = {X 416.0347, Y 44.1982, Z -1.3333, A 0.000, B 0.000, C 0.000 }
gfCNCPoint1[1878] = {X 416.0347, Y 44.9999, Z -1.3333, A 0.000, B 0.000, C 0.000 }
gfCNCPoint1[1879] = {X 416.0201, Y 45.4609, Z -1.3333, A 0.000, B 0.000, C 0.000 }
gfCNCPoint1[1880] = {X 415.9763, Y 45.9200, Z -1.3333, A 0.000, B 0.000, C 0.000 }
gfCNCPoint1[1881] = {X 419.4886, Y 45.9200, Z -1.3333, A 0.000, B 0.000, C 0.000 }
gfCNCPoint1[1882] = {X 420.8957, Y 46.0022, Z -1.3333, A 0.000, B 0.000, C 0.000 }
gfCNCPoint1[1883] = {X 422.2836, Y 46.2478, Z -1.3333, A 0.000, B 0.000, C 0.000 }
gfCNCPoint1[1884] = {X 423.4822, Y 46.5992, Z -1.3333, A 0.000, B 0.000, C 0.000 }
gfCNCPoint1[1885] = {X 424.6380, Y 47.0725, Z -1.3333, A 0.000, B 0.000, C 0.000 }
gfCNCPoint1[1886] = {X 425.7388, Y 47.6626, Z -1.3333, A 0.000, B 0.000, C 0.000 }
gfCNCPoint1[1887] = {X 425.4600, Y 46.7984, Z -1.3333, A 0.000, B 0.000, C 0.000 }
gfCNCPoint1[1888] = {X 425.2910, Y 45.9063, Z -1.3333, A 0.000, B 0.000, C 0.000 }
gfCNCPoint1[1889] = {X 425.2344, Y 45.0000, Z -1.3333, A 0.000, B 0.000, C 0.000 }
gfCNCPoint1[1890] = {X 425.2344, Y 44.2090, Z -1.3333, A 0.000, B 0.000, C 0.000 }
gfCNCPoint1[1891] = {X 425.2353, Y 44.0976, Z -1.3333, A 0.000, B 0.000, C 0.000 }
gfCNCPoint1[1892] = {X 425.2378, Y 43.9863, Z -1.3333, A 0.000, B 0.000, C 0.000 }
gfCNCPoint1[1893] = {X 425.3770, Y 42.7748, Z -1.3333, A 0.000, B 0.000, C 0.000 }
gfCNCPoint1[1894] = {X 425.7165, Y 41.6036, Z -1.3333, A 0.000, B 0.000, C 0.000 }
gfCNCPoint1[1895] = {X 426.2468, Y 40.5054, Z -1.3333, A 0.000, B 0.000, C 0.000 }
gfCNCPoint1[1896] = {X 426.9528, Y 39.5112, Z -1.3333, A 0.000, B 0.000, C 0.000 }
gfCNCPoint1[1897] = {X 427.8150, Y 38.6488, Z -1.3333, A 0.000, B 0.000, C 0.000 }
gfCNCPoint1[1898] = {X 428.8090, Y 37.9424, Z -1.3333, A 0.000, B 0.000, C 0.000 }
gfCNCPoint1[1899] = {X 431.2073, Y 33.2480, Z -1.3333, A 0.000, B 0.000, C 0.000 }
gfCNCPoint1[1900] = {X 430.0936, Y 32.1402, Z -1.3333, A 0.000, B 0.000, C 0.000 }
gfCNCPoint1[1901] = {X 429.1084, Y 30.9168, Z -1.3333, A 0.000, B 0.000, C 0.000 }
gfCNCPoint1[1902] = {X 428.2636, Y 29.5926, Z -1.3333, A 0.000, B 0.000, C 0.000 }
gfCNCPoint1[1903] = {X 427.5692, Y 28.1836, Z -1.3333, A 0.000, B 0.000, C 0.000 }
gfCNCPoint1[1904] = {X 427.0339, Y 26.7069, Z -1.3333, A 0.000, B 0.000, C 0.000 }
gfCNCPoint1[1905] = {X 426.6498, Y 25.1619, Z -1.3333, A 0.000, B 0.000, C 0.000 }
gfCNCPoint1[1906] = {X 426.3928, Y 23.5907, Z -1.3333, A 0.000, B 0.000, C 0.000 }
gfCNCPoint1[1907] = {X 426.2646, Y 22.0039, Z -1.3333, A 0.000, B 0.000, C 0.000 }
gfCNCPoint1[1908] = {X 426.2915, Y 19.9386, Z -1.3333, A 0.000, B 0.000, C 0.000 }
gfCNCPoint1[1909] = {X 426.5363, Y 17.8877, Z -1.3333, A 0.000, B 0.000, C 0.000 }
gfCNCPoint1[1910] = {X 426.9962, Y 15.8741, Z -1.3333, A 0.000, B 0.000, C 0.000 }
gfCNCPoint1[1911] = {X 427.6137, Y 14.1182, Z -1.3333, A 0.000, B 0.000, C 0.000 }
gfCNCPoint1[1912] = {X 428.4473, Y 12.4541, Z -1.3333, A 0.000, B 0.000, C 0.000 }
gfCNCPoint1[1913] = {X 429.4839, Y 10.9082, Z -1.3333, A 0.000, B 0.000, C 0.000 }
gfCNCPoint1[1914] = {X 430.7069, Y 9.5051, Z -1.3333, A 0.000, B 0.000, C 0.000 }
gfCNCPoint1[1915] = {X 426.0925, Y 9.5051, Z -1.3333, A 0.000, B 0.000, C 0.000 }
gfCNCPoint1[1916] = {X 426.3754, Y 10.3751, Z -1.3333, A 0.000, B 0.000, C 0.000 }
gfCNCPoint1[1917] = {X 426.5470, Y 11.2738, Z -1.3333, A 0.000, B 0.000, C 0.000 }
gfCNCPoint1[1918] = {X 426.6045, Y 12.1868, Z -1.3333, A 0.000, B 0.000, C 0.000 }
gfCNCPoint1[1919] = {X 426.6044, Y 12.9940, Z -1.3333, A 0.000, B 0.000, C 0.000 }
gfCNCPoint1[1920] = {X 426.4796, Y 14.2942, Z -1.3333, A 0.000, B 0.000, C 0.000 }
gfCNCPoint1[1921] = {X 426.1266, Y 15.5517, Z -1.3333, A 0.000, B 0.000, C 0.000 }
gfCNCPoint1[1922] = {X 425.5565, Y 16.7269, Z -1.3333, A 0.000, B 0.000, C 0.000 }
gfCNCPoint1[1923] = {X 424.7874, Y 17.7826, Z -1.3333, A 0.000, B 0.000, C 0.000 }
gfCNCPoint1[1924] = {X 423.8435, Y 18.6854, Z -1.3333, A 0.000, B 0.000, C 0.000 }
gfCNCPoint1[1925] = {X 422.7547, Y 19.4069, Z -1.3333, A 0.000, B 0.000, C 0.000 }
gfCNCPoint1[1926] = {X 422.3644, Y 19.9716, Z -1.3333, A 0.000, B 0.000, C 0.000 }
gfCNCPoint1[1927] = {X 422.0013, Y 20.5541, Z -1.3333, A 0.000, B 0.000, C 0.000 }
gfCNCPoint1[1928] = {X 416.2013, Y 29.8828, Z -1.3333, A 0.000, B 0.000, C 0.000 }
gfCNCPoint1[1929] = {X 414.1631, Y 28.6156, Z -1.3333, A 0.000, B 0.000, C 0.000 }
gfCNCPoint1[1930] = {X 412.1057, Y 31.9248, Z -1.3333, A 0.000, B 0.000, C 0.000 }
gfCNCPoint1[1931] = {X 412.1064, Y 40.6524, Z -1.3333, A 0.000, B 0.000, C 0.000 }
gfCNCPoint1[1932] = {X 412.7481, Y 41.4089, Z -1.3333, A 0.000, B 0.000, C 0.000 }
gfCNCPoint1[1933] = {X 413.2281, Y 42.2770, Z -1.3333, A 0.000, B 0.000, C 0.000 }
gfCNCPoint1[1934] = {X 413.5276, Y 43.2227, Z -1.3333, A 0.000, B 0.000, C 0.000 }
gfCNCPoint1[1935] = {X 413.6347, Y 44.2089, Z -1.3333, A 0.000, B 0.000, C 0.000 }
gfCNCPoint1[1936] = {X 413.6347, Y 45.0000, Z -1.3333, A 0.000, B 0.000, C 0.000 }
gfCNCPoint1[1937] = {X 413.6249, Y 45.3089, Z -1.3333, A 0.000, B 0.000, C 0.000 }
gfCNCPoint1[1938] = {X 413.5956, Y 45.6167, Z -1.3333, A 0.000, B 0.000, C 0.000 }
gfCNCPoint1[1939] = {X 413.3652, Y 46.5992, Z -1.3333, A 0.000, B 0.000, C 0.000 }
gfCNCPoint1[1940] = {X 412.9377, Y 47.5134, Z -1.3333, A 0.000, B 0.000, C 0.000 }
gfCNCPoint1[1941] = {X 412.3313, Y 48.3200, Z -1.3333, A 0.000, B 0.000, C 0.000 }
gfCNCPoint1[1942] = {X 411.9795, Y 47.9934, Z -1.3333, A 0.000, B 0.000, C 0.000 }
gfCNCPoint1[1943] = {X 411.3003, Y 48.5889, Z -1.3333, A 0.000, B 0.000, C 0.000 }
gfCNCPoint1[1944] = {X 410.5138, Y 49.0331, Z -1.3333, A 0.000, B 0.000, C 0.000 }
gfCNCPoint1[1945] = {X 409.6532, Y 49.3073, Z -1.3333, A 0.000, B 0.000, C 0.000 }
gfCNCPoint1[1946] = {X 408.7547, Y 49.4000, Z -1.3333, A 0.000, B 0.000, C 0.000 }
gfCNCPoint1[1947] = {X 402.3112, Y 49.4000, Z -1.3333, A 0.000, B 0.000, C 0.000 }
gfCNCPoint1[1948] = {X 401.3321, Y 49.2897, Z -1.3333, A 0.000, B 0.000, C 0.000 }
gfCNCPoint1[1949] = {X 400.4021, Y 48.9643, Z -1.3333, A 0.000, B 0.000, C 0.000 }
gfCNCPoint1[1950] = {X 399.5678, Y 48.4400, Z -1.3333, A 0.000, B 0.000, C 0.000 }
gfCNCPoint1[1951] = {X 398.8711, Y 47.7433, Z -1.3333, A 0.000, B 0.000, C 0.000 }
gfCNCPoint1[1952] = {X 398.3469, Y 46.9091, Z -1.3333, A 0.000, B 0.000, C 0.000 }
gfCNCPoint1[1953] = {X 398.0215, Y 45.9790, Z -1.3333, A 0.000, B 0.000, C 0.000 }
gfCNCPoint1[1954] = {X 397.9112, Y 44.9999, Z -1.3333, A 0.000, B 0.000, C 0.000 }
gfCNCPoint1[1955] = {X 397.9116, Y 44.1518, Z -1.3333, A 0.000, B 0.000, C 0.000 }
gfCNCPoint1[1956] = {X 398.0215, Y 43.2300, Z -1.3333, A 0.000, B 0.000, C 0.000 }
gfCNCPoint1[1957] = {X 398.3223, Y 42.3519, Z -1.3333, A 0.000, B 0.000, C 0.000 }
gfCNCPoint1[1958] = {X 398.8006, Y 41.5563, Z -1.3333, A 0.000, B 0.000, C 0.000 }
gfCNCPoint1[1959] = {X 399.4352, Y 40.8789, Z -1.3333, A 0.000, B 0.000, C 0.000 }
gfCNCPoint1[1960] = {X 399.4352, Y 31.6927, Z -1.3333, A 0.000, B 0.000, C 0.000 }
gfCNCPoint1[1961] = {X 393.2856, Y 20.9992, Z -1.3333, A 0.000, B 0.000, C 0.000 }
gfCNCPoint1[1962] = {X 392.4534, Y 19.5890, Z -1.3333, A 0.000, B 0.000, C 0.000 }
gfCNCPoint1[1963] = {X 391.5897, Y 18.1979, Z -1.3333, A 0.000, B 0.000, C 0.000 }
gfCNCPoint1[1964] = {X 391.1434, Y 17.5855, Z -1.3333, A 0.000, B 0.000, C 0.000 }
gfCNCPoint1[1965] = {X 390.6239, Y 17.0339, Z -1.3333, A 0.000, B 0.000, C 0.000 }
gfCNCPoint1[1966] = {X 389.8686, Y 16.6254, Z -1.3333, A 0.000, B 0.000, C 0.000 }
gfCNCPoint1[1967] = {X 389.2071, Y 16.0780, Z -1.3333, A 0.000, B 0.000, C 0.000 }
gfCNCPoint1[1968] = {X 388.6645, Y 15.4126, Z -1.3333, A 0.000, B 0.000, C 0.000 }
gfCNCPoint1[1969] = {X 388.2615, Y 14.6544, Z -1.3333, A 0.000, B 0.000, C 0.000 }
gfCNCPoint1[1970] = {X 388.0134, Y 13.8324, Z -1.3333, A 0.000, B 0.000, C 0.000 }
gfCNCPoint1[1971] = {X 387.9296, Y 12.9779, Z -1.3333, A 0.000, B 0.000, C 0.000 }
gfCNCPoint1[1972] = {X 387.9296, Y 12.1868, Z -1.3333, A 0.000, B 0.000, C 0.000 }
gfCNCPoint1[1973] = {X 388.0399, Y 11.2077, Z -1.3333, A 0.000, B 0.000, C 0.000 }
gfCNCPoint1[1974] = {X 388.3654, Y 10.2777, Z -1.3333, A 0.000, B 0.000, C 0.000 }
gfCNCPoint1[1975] = {X 388.8896, Y 9.4435, Z -1.3333, A 0.000, B 0.000, C 0.000 }
gfCNCPoint1[1976] = {X 389.5863, Y 8.7468, Z -1.3333, A 0.000, B 0.000, C 0.000 }
gfCNCPoint1[1977] = {X 390.4205, Y 8.2226, Z -1.3333, A 0.000, B 0.000, C 0.000 }
gfCNCPoint1[1978] = {X 391.3505, Y 7.8971, Z -1.3333, A 0.000, B 0.000, C 0.000 }
gfCNCPoint1[1979] = {X 392.3296, Y 7.7868, Z -1.3333, A 0.000, B 0.000, C 0.000 }
gfCNCPoint1[1980] = {X 399.1118, Y 7.7868, Z -1.3333, A 0.000, B 0.000, C 0.000 }
gfCNCPoint1[1981] = {X 400.0909, Y 7.8971, Z -1.3333, A 0.000, B 0.000, C 0.000 }
gfCNCPoint1[1982] = {X 401.0208, Y 8.2226, Z -1.3333, A 0.000, B 0.000, C 0.000 }
gfCNCPoint1[1983] = {X 401.8551, Y 8.7468, Z -1.3333, A 0.000, B 0.000, C 0.000 }
gfCNCPoint1[1984] = {X 402.5518, Y 9.4435, Z -1.3333, A 0.000, B 0.000, C 0.000 }
gfCNCPoint1[1985] = {X 403.0760, Y 10.2777, Z -1.3333, A 0.000, B 0.000, C 0.000 }
gfCNCPoint1[1986] = {X 403.4014, Y 11.2077, Z -1.3333, A 0.000, B 0.000, C 0.000 }
gfCNCPoint1[1987] = {X 403.5118, Y 12.1868, Z -1.3333, A 0.000, B 0.000, C 0.000 }
gfCNCPoint1[1988] = {X 403.5115, Y 13.0233, Z -1.3333, A 0.000, B 0.000, C 0.000 }
gfCNCPoint1[1989] = {X 403.4070, Y 13.9326, Z -1.3333, A 0.000, B 0.000, C 0.000 }
gfCNCPoint1[1990] = {X 403.1165, Y 14.8007, Z -1.3333, A 0.000, B 0.000, C 0.000 }
gfCNCPoint1[1991] = {X 405.3512, Y 18.6809, Z -1.3333, A 0.000, B 0.000, C 0.000 }
gfCNCPoint1[1992] = {X 407.7815, Y 14.7441, Z -1.3333, A 0.000, B 0.000, C 0.000 }
gfCNCPoint1[1993] = {X 407.5050, Y 13.8802, Z -1.3333, A 0.000, B 0.000, C 0.000 }
gfCNCPoint1[1994] = {X 407.4115, Y 12.9779, Z -1.3333, A 0.000, B 0.000, C 0.000 }
gfCNCPoint1[1995] = {X 407.4115, Y 12.1868, Z -1.3333, A 0.000, B 0.000, C 0.000 }
gfCNCPoint1[1996] = {X 407.5219, Y 11.2077, Z -1.3333, A 0.000, B 0.000, C 0.000 }
gfCNCPoint1[1997] = {X 407.8473, Y 10.2777, Z -1.3333, A 0.000, B 0.000, C 0.000 }
gfCNCPoint1[1998] = {X 408.3715, Y 9.4435, Z -1.3333, A 0.000, B 0.000, C 0.000 }
gfCNCPoint1[1999] = {X 409.0682, Y 8.7468, Z -1.3333, A 0.000, B 0.000, C 0.000 }
gfCNCPoint1[2000] = {X 409.9025, Y 8.2226, Z -1.3333, A 0.000, B 0.000, C 0.000 }
gfCNCPoint1[2001] = {X 410.8324, Y 7.8971, Z -1.3333, A 0.000, B 0.000, C 0.000 }
gfCNCPoint1[2002] = {X 411.8115, Y 7.7868, Z -1.3333, A 0.000, B 0.000, C 0.000 }
gfCNCPoint1[2003] = {X 419.3245, Y 7.7868, Z -1.3333, A 0.000, B 0.000, C 0.000 }
gfCNCPoint1[2004] = {X 420.3036, Y 7.8971, Z -1.3333, A 0.000, B 0.000, C 0.000 }
gfCNCPoint1[2005] = {X 421.2335, Y 8.2226, Z -1.3333, A 0.000, B 0.000, C 0.000 }
gfCNCPoint1[2006] = {X 422.0678, Y 8.7468, Z -1.3333, A 0.000, B 0.000, C 0.000 }
gfCNCPoint1[2007] = {X 422.7645, Y 9.4435, Z -1.3333, A 0.000, B 0.000, C 0.000 }
gfCNCPoint1[2008] = {X 423.2887, Y 10.2777, Z -1.3333, A 0.000, B 0.000, C 0.000 }
gfCNCPoint1[2009] = {X 423.6141, Y 11.2077, Z -1.3333, A 0.000, B 0.000, C 0.000 }
gfCNCPoint1[2010] = {X 423.7245, Y 12.1868, Z -1.3333, A 0.000, B 0.000, C 0.000 }
gfCNCPoint1[2011] = {X 423.7244, Y 12.9812, Z -1.3333, A 0.000, B 0.000, C 0.000 }
gfCNCPoint1[2012] = {X 423.6299, Y 13.8599, Z -1.3333, A 0.000, B 0.000, C 0.000 }
gfCNCPoint1[2013] = {X 423.3642, Y 14.7028, Z -1.3333, A 0.000, B 0.000, C 0.000 }
gfCNCPoint1[2014] = {X 422.9379, Y 15.4769, Z -1.3333, A 0.000, B 0.000, C 0.000 }
gfCNCPoint1[2015] = {X 422.3675, Y 16.1520, Z -1.3333, A 0.000, B 0.000, C 0.000 }
gfCNCPoint1[2016] = {X 421.6755, Y 16.7016, Z -1.3333, A 0.000, B 0.000, C 0.000 }
gfCNCPoint1[2017] = {X 420.8888, Y 17.1042, Z -1.3333, A 0.000, B 0.000, C 0.000 }
gfCNCPoint1[2018] = {X 420.1819, Y 18.0570, Z -1.3333, A 0.000, B 0.000, C 0.000 }
gfCNCPoint1[2019] = {X 419.5415, Y 19.0558, Z -1.3333, A 0.000, B 0.000, C 0.000 }
gfCNCPoint1[2020] = {X 418.0618, Y 21.4525, Z -1.3333, A 0.000, B 0.000, C 0.000 }
gfCNCPoint1[2021] = {X 411.6257, Y 31.7876, Z -1.3333, A 0.000, B 0.000, C 0.000 }
gfCNCPoint1[2022] = {X 411.6264, Y 40.8623, Z -1.3333, A 0.000, B 0.000, C 0.000 }
gfCNCPoint1[2023] = {X 412.2654, Y 41.5590, Z -1.3333, A 0.000, B 0.000, C 0.000 }
gfCNCPoint1[2024] = {X 412.7459, Y 42.3733, Z -1.3333, A 0.000, B 0.000, C 0.000 }
gfCNCPoint1[2025] = {X 413.0466, Y 43.2697, Z -1.3333, A 0.000, B 0.000, C 0.000 }
gfCNCPoint1[2026] = {X 413.1547, Y 44.2089, Z -1.3333, A 0.000, B 0.000, C 0.000 }
gfCNCPoint1[2027] = {X 413.1545, Y 45.0423, Z -1.3333, A 0.000, B 0.000, C 0.000 }
gfCNCPoint1[2028] = {X 413.0719, Y 45.8494, Z -1.3333, A 0.000, B 0.000, C 0.000 }
gfCNCPoint1[2029] = {X 412.8426, Y 46.6276, Z -1.3333, A 0.000, B 0.000, C 0.000 }
gfCNCPoint1[2030] = {X 412.4743, Y 47.3505, Z -1.3333, A 0.000, B 0.000, C 0.000 }
gfCNCPoint1[2031] = {X 411.9795, Y 47.9934, Z -1.3333, A 0.000, B 0.000, C 0.000 }
gfCNCPoint1[2032] = {X 412.3313, Y 48.3200, Z -1.3333, A 0.000, B 0.000, C 0.000 }
gfCNCPoint1[2033] = {X 419.4886, Y 48.3200, Z -1.3333, A 0.000, B 0.000, C 0.000 }
gfCNCPoint1[2034] = {X 420.8006, Y 48.4093, Z -1.3333, A 0.000, B 0.000, C 0.000 }
gfCNCPoint1[2035] = {X 422.0883, Y 48.6756, Z -1.3333, A 0.000, B 0.000, C 0.000 }
gfCNCPoint1[2036] = {X 423.3281, Y 49.1140, Z -1.3333, A 0.000, B 0.000, C 0.000 }
gfCNCPoint1[2037] = {X 424.4970, Y 49.7164, Z -1.3333, A 0.000, B 0.000, C 0.000 }
gfCNCPoint1[2038] = {X 425.4625, Y 50.3832, Z -1.3333, A 0.000, B 0.000, C 0.000 }
gfCNCPoint1[2039] = {X 426.3402, Y 51.1620, Z -1.3333, A 0.000, B 0.000, C 0.000 }
gfCNCPoint1[2040] = {X 427.1172, Y 52.0412, Z -1.3333, A 0.000, B 0.000, C 0.000 }
gfCNCPoint1[2041] = {X 427.7821, Y 53.0080, Z -1.3333, A 0.000, B 0.000, C 0.000 }
gfCNCPoint1[2042] = {X 428.1270, Y 53.6319, Z -1.3333, A 0.000, B 0.000, C 0.000 }
gfCNCPoint1[2043] = {X 428.4251, Y 54.2795, Z -1.3333, A 0.000, B 0.000, C 0.000 }
gfCNCPoint1[2044] = {X 431.5821, Y 55.5101, Z -1.3333, A 0.000, B 0.000, C 0.000 }
gfCNCPoint1[2045] = {X 449.5100, Y 62.6228, Z -1.3333, A 0.000, B 0.000, C 0.000 }
gfCNCPoint1[2046] = {X 449.1116, Y 61.4475, Z -1.3333, A 0.000, B 0.000, C 0.000 }
gfCNCPoint1[2047] = {X 448.8669, Y 60.2309, Z -1.3333, A 0.000, B 0.000, C 0.000 }
gfCNCPoint1[2048] = {X 448.7798, Y 58.9930, Z -1.3333, A 0.000, B 0.000, C 0.000 }
gfCNCPoint1[2049] = {X 448.7796, Y 58.0000, Z -1.3333, A 0.000, B 0.000, C 0.000 }
gfCNCPoint1[2050] = {X 448.8564, Y 56.7833, Z -1.3333, A 0.000, B 0.000, C 0.000 }
gfCNCPoint1[2051] = {X 449.0855, Y 55.5859, Z -1.3333, A 0.000, B 0.000, C 0.000 }
gfCNCPoint1[2052] = {X 449.4632, Y 54.4268, Z -1.3333, A 0.000, B 0.000, C 0.000 }
gfCNCPoint1[2053] = {X 449.9837, Y 53.3244, Z -1.3333, A 0.000, B 0.000, C 0.000 }
gfCNCPoint1[2054] = {X 450.6386, Y 52.2961, Z -1.3333, A 0.000, B 0.000, C 0.000 }
gfCNCPoint1[2055] = {X 451.3887, Y 51.3890, Z -1.3333, A 0.000, B 0.000, C 0.000 }
gfCNCPoint1[2056] = {X 452.2434, Y 50.5796, Z -1.3333, A 0.000, B 0.000, C 0.000 }
gfCNCPoint1[2057] = {X 453.1901, Y 49.8800, Z -1.3333, A 0.000, B 0.000, C 0.000 }
gfCNCPoint1[2058] = {X 452.3731, Y 49.8442, Z -1.3333, A 0.000, B 0.000, C 0.000 }
gfCNCPoint1[2059] = {X 451.5735, Y 49.6724, Z -1.3333, A 0.000, B 0.000, C 0.000 }
gfCNCPoint1[2060] = {X 450.8138, Y 49.3696, Z -1.3333, A 0.000, B 0.000, C 0.000 }
gfCNCPoint1[2061] = {X 450.1154, Y 48.9441, Z -1.3333, A 0.000, B 0.000, C 0.000 }
gfCNCPoint1[2062] = {X 449.3503, Y 48.2496, Z -1.3333, A 0.000, B 0.000, C 0.000 }
gfCNCPoint1[2063] = {X 448.7486, Y 47.4095, Z -1.3333, A 0.000, B 0.000, C 0.000 }
gfCNCPoint1[2064] = {X 448.3373, Y 46.4616, Z -1.3333, A 0.000, B 0.000, C 0.000 }
gfCNCPoint1[2065] = {X 448.1732, Y 45.7588, Z -1.3333, A 0.000, B 0.000, C 0.000 }
gfCNCPoint1[2066] = {X 448.1146, Y 45.0395, Z -1.3333, A 0.000, B 0.000, C 0.000 }
gfCNCPoint1[2067] = {X 448.1149, Y 44.1417, Z -1.3333, A 0.000, B 0.000, C 0.000 }
gfCNCPoint1[2068] = {X 448.2252, Y 43.1751, Z -1.3333, A 0.000, B 0.000, C 0.000 }
gfCNCPoint1[2069] = {X 448.5250, Y 42.2497, Z -1.3333, A 0.000, B 0.000, C 0.000 }
gfCNCPoint1[2070] = {X 449.0024, Y 41.4021, Z -1.3333, A 0.000, B 0.000, C 0.000 }
gfCNCPoint1[2071] = {X 449.6384, Y 40.6660, Z -1.3333, A 0.000, B 0.000, C 0.000 }
gfCNCPoint1[2072] = {X 449.6384, Y 35.0338, Z -1.3333, A 0.000, B 0.000, C 0.000 }
gfCNCPoint1[2073] = {X 447.8153, Y 35.0338, Z -1.3333, A 0.000, B 0.000, C 0.000 }
gfCNCPoint1[2074] = {X 443.7922, Y 42.8665, Z -1.3333, A 0.000, B 0.000, C 0.000 }
gfCNCPoint1[2075] = {X 443.9301, Y 43.5096, Z -1.3333, A 0.000, B 0.000, C 0.000 }
gfCNCPoint1[2076] = {X 443.9803, Y 44.1653, Z -1.3333, A 0.000, B 0.000, C 0.000 }
gfCNCPoint1[2077] = {X 443.9805, Y 45.0000, Z -1.3333, A 0.000, B 0.000, C 0.000 }
gfCNCPoint1[2078] = {X 443.9242, Y 45.7387, Z -1.3333, A 0.000, B 0.000, C 0.000 }
gfCNCPoint1[2079] = {X 443.7568, Y 46.4603, Z -1.3333, A 0.000, B 0.000, C 0.000 }
gfCNCPoint1[2080] = {X 443.3736, Y 47.3569, Z -1.3333, A 0.000, B 0.000, C 0.000 }
gfCNCPoint1[2081] = {X 442.8197, Y 48.1594, Z -1.3333, A 0.000, B 0.000, C 0.000 }
gfCNCPoint1[2082] = {X 442.1173, Y 48.8357, Z -1.3333, A 0.000, B 0.000, C 0.000 }
gfCNCPoint1[2083] = {X 441.2945, Y 49.3590, Z -1.3333, A 0.000, B 0.000, C 0.000 }
gfCNCPoint1[2084] = {X 440.3841, Y 49.7081, Z -1.3333, A 0.000, B 0.000, C 0.000 }
gfCNCPoint1[2085] = {X 441.6467, Y 54.3391, Z -1.3333, A 0.000, B 0.000, C 0.000 }
gfCNCPoint1[2086] = {X 444.2221, Y 55.3609, Z -1.3333, A 0.000, B 0.000, C 0.000 }
gfCNCPoint1[2087] = {X 444.5424, Y 54.0022, Z -1.3333, A 0.000, B 0.000, C 0.000 }
gfCNCPoint1[2088] = {X 444.9921, Y 52.6806, Z -1.3333, A 0.000, B 0.000, C 0.000 }
gfCNCPoint1[2089] = {X 443.9518, Y 53.3766, Z -1.3333, A 0.000, B 0.000, C 0.000 }
gfCNCPoint1[2090] = {X 442.8304, Y 53.9325, Z -1.3333, A 0.000, B 0.000, C 0.000 }
gfCNCPoint1[2091] = {X 441.6467, Y 54.3391, Z -1.3333, A 0.000, B 0.000, C 0.000 }
gfCNCPoint1[2092] = {X 441.0154, Y 52.0236, Z -1.3333, A 0.000, B 0.000, C 0.000 }
gfCNCPoint1[2093] = {X 440.0665, Y 52.2156, Z -1.3333, A 0.000, B 0.000, C 0.000 }
gfCNCPoint1[2094] = {X 439.1005, Y 52.2800, Z -1.3333, A 0.000, B 0.000, C 0.000 }
gfCNCPoint1[2095] = {X 432.5144, Y 52.2800, Z -1.3333, A 0.000, B 0.000, C 0.000 }
gfCNCPoint1[2096] = {X 431.6034, Y 52.2228, Z -1.3333, A 0.000, B 0.000, C 0.000 }
gfCNCPoint1[2097] = {X 430.7066, Y 52.0520, Z -1.3333, A 0.000, B 0.000, C 0.000 }
gfCNCPoint1[2098] = {X 429.8384, Y 51.7703, Z -1.3333, A 0.000, B 0.000, C 0.000 }
gfCNCPoint1[2099] = {X 430.0173, Y 52.0778, Z -1.3333, A 0.000, B 0.000, C 0.000 }
gfCNCPoint1[2100] = {X 430.1872, Y 52.3904, Z -1.3333, A 0.000, B 0.000, C 0.000 }
gfCNCPoint1[2101] = {X 432.4637, Y 53.2778, Z -1.3333, A 0.000, B 0.000, C 0.000 }
gfCNCPoint1[2102] = {X 446.3797, Y 58.7989, Z -1.3333, A 0.000, B 0.000, C 0.000 }
gfCNCPoint1[2103] = {X 446.3796, Y 58.0000, Z -1.3333, A 0.000, B 0.000, C 0.000 }
gfCNCPoint1[2104] = {X 446.4303, Y 56.8945, Z -1.3333, A 0.000, B 0.000, C 0.000 }
gfCNCPoint1[2105] = {X 446.5819, Y 55.7983, Z -1.3333, A 0.000, B 0.000, C 0.000 }
gfCNCPoint1[2106] = {X 446.8491, Y 54.6648, Z -1.3333, A 0.000, B 0.000, C 0.000 }
gfCNCPoint1[2107] = {X 447.2243, Y 53.5622, Z -1.3333, A 0.000, B 0.000, C 0.000 }
gfCNCPoint1[2108] = {X 447.8767, Y 52.1752, Z -1.3333, A 0.000, B 0.000, C 0.000 }
gfCNCPoint1[2109] = {X 448.6995, Y 50.8820, Z -1.3333, A 0.000, B 0.000, C 0.000 }
gfCNCPoint1[2110] = {X 447.8224, Y 50.1272, Z -1.3333, A 0.000, B 0.000, C 0.000 }
gfCNCPoint1[2111] = {X 447.0760, Y 49.2431, Z -1.3333, A 0.000, B 0.000, C 0.000 }
gfCNCPoint1[2112] = {X 446.4792, Y 48.2518, Z -1.3333, A 0.000, B 0.000, C 0.000 }
gfCNCPoint1[2113] = {X 446.0469, Y 47.1785, Z -1.3333, A 0.000, B 0.000, C 0.000 }
gfCNCPoint1[2114] = {X 445.6333, Y 48.2126, Z -1.3333, A 0.000, B 0.000, C 0.000 }
gfCNCPoint1[2115] = {X 445.0668, Y 49.1715, Z -1.3333, A 0.000, B 0.000, C 0.000 }
gfCNCPoint1[2116] = {X 444.3606, Y 50.0328, Z -1.3333, A 0.000, B 0.000, C 0.000 }
gfCNCPoint1[2117] = {X 443.5314, Y 50.7763, Z -1.3333, A 0.000, B 0.000, C 0.000 }
gfCNCPoint1[2118] = {X 442.7490, Y 51.2997, Z -1.3333, A 0.000, B 0.000, C 0.000 }
gfCNCPoint1[2119] = {X 441.9056, Y 51.7178, Z -1.3333, A 0.000, B 0.000, C 0.000 }
gfCNCPoint1[2120] = {X 441.0154, Y 52.0236, Z -1.3333, A 0.000, B 0.000, C 0.000 }
gfCNCPoint1[2121] = {X 440.3841, Y 49.7081, Z -1.3333, A 0.000, B 0.000, C 0.000 }
gfCNCPoint1[2122] = {X 439.7480, Y 49.8368, Z -1.3333, A 0.000, B 0.000, C 0.000 }
gfCNCPoint1[2123] = {X 439.1005, Y 49.8800, Z -1.3333, A 0.000, B 0.000, C 0.000 }
gfCNCPoint1[2124] = {X 432.5144, Y 49.8800, Z -1.3333, A 0.000, B 0.000, C 0.000 }
gfCNCPoint1[2125] = {X 431.6014, Y 49.7938, Z -1.3333, A 0.000, B 0.000, C 0.000 }
gfCNCPoint1[2126] = {X 430.7206, Y 49.5383, Z -1.3333, A 0.000, B 0.000, C 0.000 }
gfCNCPoint1[2127] = {X 429.8343, Y 49.0782, Z -1.3333, A 0.000, B 0.000, C 0.000 }
gfCNCPoint1[2128] = {X 429.0603, Y 48.4473, Z -1.3333, A 0.000, B 0.000, C 0.000 }
gfCNCPoint1[2129] = {X 428.4309, Y 47.6720, Z -1.3333, A 0.000, B 0.000, C 0.000 }
gfCNCPoint1[2130] = {X 427.9725, Y 46.7848, Z -1.3333, A 0.000, B 0.000, C 0.000 }
gfCNCPoint1[2131] = {X 427.7197, Y 45.9083, Z -1.3333, A 0.000, B 0.000, C 0.000 }
gfCNCPoint1[2132] = {X 427.6344, Y 45.0000, Z -1.3333, A 0.000, B 0.000, C 0.000 }
gfCNCPoint1[2133] = {X 427.6344, Y 44.2089, Z -1.3333, A 0.000, B 0.000, C 0.000 }
gfCNCPoint1[2134] = {X 427.7263, Y 43.2661, Z -1.3333, A 0.000, B 0.000, C 0.000 }
gfCNCPoint1[2135] = {X 427.9987, Y 42.3588, Z -1.3333, A 0.000, B 0.000, C 0.000 }
gfCNCPoint1[2136] = {X 428.4411, Y 41.5213, Z -1.3333, A 0.000, B 0.000, C 0.000 }
gfCNCPoint1[2137] = {X 429.0371, Y 40.7849, Z -1.3333, A 0.000, B 0.000, C 0.000 }
gfCNCPoint1[2138] = {X 429.7641, Y 40.1776, Z -1.3333, A 0.000, B 0.000, C 0.000 }
gfCNCPoint1[2139] = {X 430.5947, Y 39.7222, Z -1.3333, A 0.000, B 0.000, C 0.000 }
gfCNCPoint1[2140] = {X 434.2536, Y 32.5604, Z -1.3333, A 0.000, B 0.000, C 0.000 }
gfCNCPoint1[2141] = {X 432.9194, Y 31.5577, Z -1.3333, A 0.000, B 0.000, C 0.000 }
gfCNCPoint1[2142] = {X 431.7389, Y 30.3779, Z -1.3333, A 0.000, B 0.000, C 0.000 }
gfCNCPoint1[2143] = {X 430.7353, Y 29.0443, Z -1.3333, A 0.000, B 0.000, C 0.000 }
gfCNCPoint1[2144] = {X 429.9286, Y 27.5832, Z -1.3333, A 0.000, B 0.000, C 0.000 }
gfCNCPoint1[2145] = {X 429.3346, Y 26.0235, Z -1.3333, A 0.000, B 0.000, C 0.000 }
gfCNCPoint1[2146] = {X 428.9005, Y 24.1500, Z -1.3333, A 0.000, B 0.000, C 0.000 }
gfCNCPoint1[2147] = {X 428.6791, Y 22.2397, Z -1.3333, A 0.000, B 0.000, C 0.000 }
gfCNCPoint1[2148] = {X 428.6732, Y 20.3165, Z -1.3333, A 0.000, B 0.000, C 0.000 }
gfCNCPoint1[2149] = {X 428.8828, Y 18.4048, Z -1.3333, A 0.000, B 0.000, C 0.000 }
gfCNCPoint1[2150] = {X 429.3053, Y 16.5287, Z -1.3333, A 0.000, B 0.000, C 0.000 }
gfCNCPoint1[2151] = {X 429.8222, Y 15.0577, Z -1.3333, A 0.000, B 0.000, C 0.000 }
gfCNCPoint1[2152] = {X 430.5203, Y 13.6635, Z -1.3333, A 0.000, B 0.000, C 0.000 }
gfCNCPoint1[2153] = {X 431.3885, Y 12.3685, Z -1.3333, A 0.000, B 0.000, C 0.000 }
gfCNCPoint1[2154] = {X 432.4130, Y 11.1931, Z -1.3333, A 0.000, B 0.000, C 0.000 }
gfCNCPoint1[2155] = {X 433.6950, Y 10.0651, Z -1.3333, A 0.000, B 0.000, C 0.000 }
gfCNCPoint1[2156] = {X 435.1204, Y 9.1247, Z -1.3333, A 0.000, B 0.000, C 0.000 }
gfCNCPoint1[2157] = {X 436.6619, Y 8.3899, Z -1.3333, A 0.000, B 0.000, C 0.000 }
gfCNCPoint1[2158] = {X 438.2899, Y 7.8747, Z -1.3333, A 0.000, B 0.000, C 0.000 }
gfCNCPoint1[2159] = {X 439.9586, Y 7.5568, Z -1.3333, A 0.000, B 0.000, C 0.000 }
gfCNCPoint1[2160] = {X 441.6470, Y 7.3701, Z -1.3333, A 0.000, B 0.000, C 0.000 }
gfCNCPoint1[2161] = {X 443.3449, Y 7.3159, Z -1.3333, A 0.000, B 0.000, C 0.000 }
gfCNCPoint1[2162] = {X 459.4465, Y 7.3119, Z -1.3333, A 0.000, B 0.000, C 0.000 }
gfCNCPoint1[2163] = {X 460.4092, Y 7.4080, Z -1.3333, A 0.000, B 0.000, C 0.000 }
gfCNCPoint1[2164] = {X 461.3339, Y 7.6924, Z -1.3333, A 0.000, B 0.000, C 0.000 }
gfCNCPoint1[2165] = {X 462.1842, Y 8.1540, Z -1.3333, A 0.000, B 0.000, C 0.000 }
gfCNCPoint1[2166] = {X 462.9265, Y 8.7745, Z -1.3333, A 0.000, B 0.000, C 0.000 }
gfCNCPoint1[2167] = {X 463.5316, Y 9.5294, Z -1.3333, A 0.000, B 0.000, C 0.000 }
gfCNCPoint1[2168] = {X 463.9755, Y 10.3891, Z -1.3333, A 0.000, B 0.000, C 0.000 }
gfCNCPoint1[2169] = {X 464.2316, Y 11.2700, Z -1.3333, A 0.000, B 0.000, C 0.000 }
gfCNCPoint1[2170] = {X 464.3179, Y 12.1834, Z -1.3333, A 0.000, B 0.000, C 0.000 }
gfCNCPoint1[2171] = {X 464.3179, Y 12.9779, Z -1.3333, A 0.000, B 0.000, C 0.000 }
gfCNCPoint1[2172] = {X 464.2173, Y 13.9639, Z -1.3333, A 0.000, B 0.000, C 0.000 }
gfCNCPoint1[2173] = {X 463.9196, Y 14.9092, Z -1.3333, A 0.000, B 0.000, C 0.000 }
gfCNCPoint1[2174] = {X 463.4370, Y 15.7748, Z -1.3333, A 0.000, B 0.000, C 0.000 }
gfCNCPoint1[2175] = {X 462.7894, Y 16.5251, Z -1.3333, A 0.000, B 0.000, C 0.000 }
gfCNCPoint1[2176] = {X 462.7898, Y 40.6621, Z -1.3333, A 0.000, B 0.000, C 0.000 }
gfCNCPoint1[2177] = {X 463.4312, Y 41.4037, Z -1.3333, A 0.000, B 0.000, C 0.000 }
gfCNCPoint1[2178] = {X 463.9113, Y 42.2586, Z -1.3333, A 0.000, B 0.000, C 0.000 }
gfCNCPoint1[2179] = {X 464.2109, Y 43.1923, Z -1.3333, A 0.000, B 0.000, C 0.000 }
gfCNCPoint1[2180] = {X 464.3178, Y 44.1670, Z -1.3333, A 0.000, B 0.000, C 0.000 }
gfCNCPoint1[2181] = {X 464.3179, Y 45.0000, Z -1.3333, A 0.000, B 0.000, C 0.000 }
gfCNCPoint1[2182] = {X 464.3081, Y 45.3090, Z -1.3333, A 0.000, B 0.000, C 0.000 }
gfCNCPoint1[2183] = {X 464.2788, Y 45.6167, Z -1.3333, A 0.000, B 0.000, C 0.000 }
gfCNCPoint1[2184] = {X 464.0485, Y 46.5992, Z -1.3333, A 0.000, B 0.000, C 0.000 }
gfCNCPoint1[2185] = {X 463.6209, Y 47.5134, Z -1.3333, A 0.000, B 0.000, C 0.000 }
gfCNCPoint1[2186] = {X 463.0145, Y 48.3200, Z -1.3333, A 0.000, B 0.000, C 0.000 }
gfCNCPoint1[2187] = {X 462.6627, Y 47.9934, Z -1.3333, A 0.000, B 0.000, C 0.000 }
gfCNCPoint1[2188] = {X 461.9835, Y 48.5889, Z -1.3333, A 0.000, B 0.000, C 0.000 }
gfCNCPoint1[2189] = {X 461.1970, Y 49.0331, Z -1.3333, A 0.000, B 0.000, C 0.000 }
gfCNCPoint1[2190] = {X 460.3364, Y 49.3073, Z -1.3333, A 0.000, B 0.000, C 0.000 }
gfCNCPoint1[2191] = {X 459.4379, Y 49.4000, Z -1.3333, A 0.000, B 0.000, C 0.000 }
gfCNCPoint1[2192] = {X 452.9945, Y 49.4000, Z -1.3333, A 0.000, B 0.000, C 0.000 }
gfCNCPoint1[2193] = {X 452.0154, Y 49.2897, Z -1.3333, A 0.000, B 0.000, C 0.000 }
gfCNCPoint1[2194] = {X 451.0854, Y 48.9643, Z -1.3333, A 0.000, B 0.000, C 0.000 }
gfCNCPoint1[2195] = {X 450.2511, Y 48.4400, Z -1.3333, A 0.000, B 0.000, C 0.000 }
gfCNCPoint1[2196] = {X 449.5544, Y 47.7433, Z -1.3333, A 0.000, B 0.000, C 0.000 }
gfCNCPoint1[2197] = {X 449.0302, Y 46.9091, Z -1.3333, A 0.000, B 0.000, C 0.000 }
gfCNCPoint1[2198] = {X 448.7048, Y 45.9790, Z -1.3333, A 0.000, B 0.000, C 0.000 }
gfCNCPoint1[2199] = {X 448.5945, Y 44.9999, Z -1.3333, A 0.000, B 0.000, C 0.000 }
gfCNCPoint1[2200] = {X 448.5949, Y 44.1483, Z -1.3333, A 0.000, B 0.000, C 0.000 }
gfCNCPoint1[2201] = {X 448.7053, Y 43.2275, Z -1.3333, A 0.000, B 0.000, C 0.000 }
gfCNCPoint1[2202] = {X 449.0063, Y 42.3503, Z -1.3333, A 0.000, B 0.000, C 0.000 }
gfCNCPoint1[2203] = {X 449.4844, Y 41.5556, Z -1.3333, A 0.000, B 0.000, C 0.000 }
gfCNCPoint1[2204] = {X 450.1184, Y 40.8789, Z -1.3333, A 0.000, B 0.000, C 0.000 }
gfCNCPoint1[2205] = {X 450.1184, Y 34.5538, Z -1.3333, A 0.000, B 0.000, C 0.000 }
gfCNCPoint1[2206] = {X 447.5222, Y 34.5538, Z -1.3333, A 0.000, B 0.000, C 0.000 }
gfCNCPoint1[2207] = {X 443.2759, Y 42.8211, Z -1.3333, A 0.000, B 0.000, C 0.000 }
gfCNCPoint1[2208] = {X 443.4440, Y 43.5060, Z -1.3333, A 0.000, B 0.000, C 0.000 }
gfCNCPoint1[2209] = {X 443.5005, Y 44.2089, Z -1.3333, A 0.000, B 0.000, C 0.000 }
gfCNCPoint1[2210] = {X 443.5005, Y 45.0000, Z -1.3333, A 0.000, B 0.000, C 0.000 }
gfCNCPoint1[2211] = {X 443.3902, Y 45.9791, Z -1.3333, A 0.000, B 0.000, C 0.000 }
gfCNCPoint1[2212] = {X 443.0647, Y 46.9091, Z -1.3333, A 0.000, B 0.000, C 0.000 }
gfCNCPoint1[2213] = {X 442.5405, Y 47.7434, Z -1.3333, A 0.000, B 0.000, C 0.000 }
gfCNCPoint1[2214] = {X 441.8438, Y 48.4401, Z -1.3333, A 0.000, B 0.000, C 0.000 }
gfCNCPoint1[2215] = {X 441.0096, Y 48.9643, Z -1.3333, A 0.000, B 0.000, C 0.000 }
gfCNCPoint1[2216] = {X 440.0796, Y 49.2897, Z -1.3333, A 0.000, B 0.000, C 0.000 }
gfCNCPoint1[2217] = {X 439.1005, Y 49.4000, Z -1.3333, A 0.000, B 0.000, C 0.000 }
gfCNCPoint1[2218] = {X 432.5144, Y 49.4000, Z -1.3333, A 0.000, B 0.000, C 0.000 }
gfCNCPoint1[2219] = {X 431.5353, Y 49.2897, Z -1.3333, A 0.000, B 0.000, C 0.000 }
gfCNCPoint1[2220] = {X 430.6053, Y 48.9643, Z -1.3333, A 0.000, B 0.000, C 0.000 }
gfCNCPoint1[2221] = {X 429.7711, Y 48.4401, Z -1.3333, A 0.000, B 0.000, C 0.000 }
gfCNCPoint1[2222] = {X 429.0743, Y 47.7434, Z -1.3333, A 0.000, B 0.000, C 0.000 }
gfCNCPoint1[2223] = {X 428.5501, Y 46.9091, Z -1.3333, A 0.000, B 0.000, C 0.000 }
gfCNCPoint1[2224] = {X 428.2247, Y 45.9791, Z -1.3333, A 0.000, B 0.000, C 0.000 }
gfCNCPoint1[2225] = {X 428.1144, Y 45.0000, Z -1.3333, A 0.000, B 0.000, C 0.000 }
gfCNCPoint1[2226] = {X 428.1148, Y 44.1483, Z -1.3333, A 0.000, B 0.000, C 0.000 }
gfCNCPoint1[2227] = {X 428.2132, Y 43.2816, Z -1.3333, A 0.000, B 0.000, C 0.000 }
gfCNCPoint1[2228] = {X 428.4806, Y 42.4514, Z -1.3333, A 0.000, B 0.000, C 0.000 }
gfCNCPoint1[2229] = {X 428.9065, Y 41.6903, Z -1.3333, A 0.000, B 0.000, C 0.000 }
gfCNCPoint1[2230] = {X 429.4741, Y 41.0281, Z -1.3333, A 0.000, B 0.000, C 0.000 }
gfCNCPoint1[2231] = {X 430.1613, Y 40.4909, Z -1.3333, A 0.000, B 0.000, C 0.000 }
gfCNCPoint1[2232] = {X 430.9408, Y 40.0998, Z -1.3333, A 0.000, B 0.000, C 0.000 }
gfCNCPoint1[2233] = {X 434.8820, Y 32.3854, Z -1.3333, A 0.000, B 0.000, C 0.000 }
gfCNCPoint1[2234] = {X 433.7186, Y 31.5929, Z -1.3333, A 0.000, B 0.000, C 0.000 }
gfCNCPoint1[2235] = {X 432.6618, Y 30.6631, Z -1.3333, A 0.000, B 0.000, C 0.000 }
gfCNCPoint1[2236] = {X 431.7276, Y 29.6101, Z -1.3333, A 0.000, B 0.000, C 0.000 }
gfCNCPoint1[2237] = {X 430.9304, Y 28.4500, Z -1.3333, A 0.000, B 0.000, C 0.000 }
gfCNCPoint1[2238] = {X 430.2821, Y 27.2005, Z -1.3333, A 0.000, B 0.000, C 0.000 }
gfCNCPoint1[2239] = {X 429.7928, Y 25.8807, Z -1.3333, A 0.000, B 0.000, C 0.000 }
gfCNCPoint1[2240] = {X 429.3722, Y 24.0610, Z -1.3333, A 0.000, B 0.000, C 0.000 }
gfCNCPoint1[2241] = {X 429.1579, Y 22.2057, Z -1.3333, A 0.000, B 0.000, C 0.000 }
gfCNCPoint1[2242] = {X 429.1527, Y 20.3381, Z -1.3333, A 0.000, B 0.000, C 0.000 }
gfCNCPoint1[2243] = {X 429.3566, Y 18.4816, Z -1.3333, A 0.000, B 0.000, C 0.000 }
gfCNCPoint1[2244] = {X 429.7670, Y 16.6596, Z -1.3333, A 0.000, B 0.000, C 0.000 }
gfCNCPoint1[2245] = {X 430.2921, Y 15.1795, Z -1.3333, A 0.000, B 0.000, C 0.000 }
gfCNCPoint1[2246] = {X 431.0081, Y 13.7816, Z -1.3333, A 0.000, B 0.000, C 0.000 }
gfCNCPoint1[2247] = {X 431.9022, Y 12.4904, Z -1.3333, A 0.000, B 0.000, C 0.000 }
gfCNCPoint1[2248] = {X 432.9590, Y 11.3286, Z -1.3333, A 0.000, B 0.000, C 0.000 }
gfCNCPoint1[2249] = {X 434.1599, Y 10.3165, Z -1.3333, A 0.000, B 0.000, C 0.000 }
gfCNCPoint1[2250] = {X 435.4839, Y 9.4717, Z -1.3333, A 0.000, B 0.000, C 0.000 }
gfCNCPoint1[2251] = {X 436.9079, Y 8.8091, Z -1.3333, A 0.000, B 0.000, C 0.000 }
gfCNCPoint1[2252] = {X 438.4068, Y 8.3403, Z -1.3333, A 0.000, B 0.000, C 0.000 }
gfCNCPoint1[2253] = {X 440.0368, Y 8.0304, Z -1.3333, A 0.000, B 0.000, C 0.000 }
gfCNCPoint1[2254] = {X 441.6861, Y 7.8486, Z -1.3333, A 0.000, B 0.000, C 0.000 }
gfCNCPoint1[2255] = {X 443.3445, Y 7.7959, Z -1.3333, A 0.000, B 0.000, C 0.000 }
gfCNCPoint1[2256] = {X 444.0367, Y 7.7919, Z -1.3333, A 0.000, B 0.000, C 0.000 }
gfCNCPoint1[2257] = {X 459.4465, Y 7.7919, Z -1.3333, A 0.000, B 0.000, C 0.000 }
gfCNCPoint1[2258] = {X 460.4237, Y 7.9020, Z -1.3333, A 0.000, B 0.000, C 0.000 }
gfCNCPoint1[2259] = {X 461.3519, Y 8.2268, Z -1.3333, A 0.000, B 0.000, C 0.000 }
gfCNCPoint1[2260] = {X 462.1845, Y 8.7500, Z -1.3333, A 0.000, B 0.000, C 0.000 }
gfCNCPoint1[2261] = {X 462.8799, Y 9.4453, Z -1.3333, A 0.000, B 0.000, C 0.000 }
gfCNCPoint1[2262] = {X 463.4031, Y 10.2780, Z -1.3333, A 0.000, B 0.000, C 0.000 }
gfCNCPoint1[2263] = {X 463.7278, Y 11.2062, Z -1.3333, A 0.000, B 0.000, C 0.000 }
gfCNCPoint1[2264] = {X 463.8379, Y 12.1834, Z -1.3333, A 0.000, B 0.000, C 0.000 }
gfCNCPoint1[2265] = {X 463.8377, Y 13.0201, Z -1.3333, A 0.000, B 0.000, C 0.000 }
gfCNCPoint1[2266] = {X 463.7298, Y 13.9473, Z -1.3333, A 0.000, B 0.000, C 0.000 }
gfCNCPoint1[2267] = {X 463.4288, Y 14.8309, Z -1.3333, A 0.000, B 0.000, C 0.000 }
gfCNCPoint1[2268] = {X 462.9481, Y 15.6311, Z -1.3333, A 0.000, B 0.000, C 0.000 }
gfCNCPoint1[2269] = {X 462.3094, Y 16.3119, Z -1.3333, A 0.000, B 0.000, C 0.000 }
gfCNCPoint1[2270] = {X 462.3098, Y 40.8753, Z -1.3333, A 0.000, B 0.000, C 0.000 }
gfCNCPoint1[2271] = {X 462.9547, Y 41.5645, Z -1.3333, A 0.000, B 0.000, C 0.000 }
gfCNCPoint1[2272] = {X 463.4377, Y 42.3753, Z -1.3333, A 0.000, B 0.000, C 0.000 }
gfCNCPoint1[2273] = {X 463.7367, Y 43.2705, Z -1.3333, A 0.000, B 0.000, C 0.000 }
gfCNCPoint1[2274] = {X 463.8379, Y 44.2089, Z -1.3333, A 0.000, B 0.000, C 0.000 }
gfCNCPoint1[2275] = {X 463.8379, Y 45.0000, Z -1.3333, A 0.000, B 0.000, C 0.000 }
gfCNCPoint1[2276] = {X 463.7612, Y 45.8182, Z -1.3333, A 0.000, B 0.000, C 0.000 }
gfCNCPoint1[2277] = {X 463.5336, Y 46.6079, Z -1.3333, A 0.000, B 0.000, C 0.000 }
gfCNCPoint1[2278] = {X 463.1632, Y 47.3415, Z -1.3333, A 0.000, B 0.000, C 0.000 }
gfCNCPoint1[2279] = {X 462.6627, Y 47.9934, Z -1.3333, A 0.000, B 0.000, C 0.000 }
gfCNCPoint1[2280] = {X 463.0145, Y 48.3200, Z -1.3333, A 0.000, B 0.000, C 0.000 }
gfCNCPoint1[2281] = {X 472.1884, Y 48.3200, Z -1.3333, A 0.000, B 0.000, C 0.000 }
gfCNCPoint1[2282] = {X 471.5820, Y 47.5134, Z -1.3333, A 0.000, B 0.000, C 0.000 }
gfCNCPoint1[2283] = {X 471.1544, Y 46.5992, Z -1.3333, A 0.000, B 0.000, C 0.000 }
gfCNCPoint1[2284] = {X 470.9241, Y 45.6167, Z -1.3333, A 0.000, B 0.000, C 0.000 }
gfCNCPoint1[2285] = {X 470.8947, Y 45.3090, Z -1.3333, A 0.000, B 0.000, C 0.000 }
gfCNCPoint1[2286] = {X 470.8850, Y 45.0000, Z -1.3333, A 0.000, B 0.000, C 0.000 }
gfCNCPoint1[2287] = {X 470.8850, Y 44.2089, Z -1.3333, A 0.000, B 0.000, C 0.000 }
gfCNCPoint1[2288] = {X 470.9769, Y 43.2661, Z -1.3333, A 0.000, B 0.000, C 0.000 }
gfCNCPoint1[2289] = {X 471.2492, Y 42.3588, Z -1.3333, A 0.000, B 0.000, C 0.000 }
gfCNCPoint1[2290] = {X 471.6917, Y 41.5213, Z -1.3333, A 0.000, B 0.000, C 0.000 }
gfCNCPoint1[2291] = {X 472.2877, Y 40.7849, Z -1.3333, A 0.000, B 0.000, C 0.000 }
gfCNCPoint1[2292] = {X 473.0146, Y 40.1776, Z -1.3333, A 0.000, B 0.000, C 0.000 }
gfCNCPoint1[2293] = {X 473.8453, Y 39.7222, Z -1.3333, A 0.000, B 0.000, C 0.000 }
gfCNCPoint1[2294] = {X 477.5004, Y 32.5677, Z -1.3333, A 0.000, B 0.000, C 0.000 }
gfCNCPoint1[2295] = {X 476.2834, Y 31.6576, Z -1.3333, A 0.000, B 0.000, C 0.000 }
gfCNCPoint1[2296] = {X 475.1908, Y 30.6014, Z -1.3333, A 0.000, B 0.000, C 0.000 }
gfCNCPoint1[2297] = {X 474.2401, Y 29.4159, Z -1.3333, A 0.000, B 0.000, C 0.000 }
gfCNCPoint1[2298] = {X 473.4464, Y 28.1199, Z -1.3333, A 0.000, B 0.000, C 0.000 }
gfCNCPoint1[2299] = {X 472.8224, Y 26.7343, Z -1.3333, A 0.000, B 0.000, C 0.000 }
gfCNCPoint1[2300] = {X 472.3781, Y 25.2811, Z -1.3333, A 0.000, B 0.000, C 0.000 }
gfCNCPoint1[2301] = {X 472.0535, Y 23.5418, Z -1.3333, A 0.000, B 0.000, C 0.000 }
gfCNCPoint1[2302] = {X 471.9083, Y 21.7784, Z -1.3333, A 0.000, B 0.000, C 0.000 }
gfCNCPoint1[2303] = {X 471.9443, Y 20.0094, Z -1.3333, A 0.000, B 0.000, C 0.000 }
gfCNCPoint1[2304] = {X 472.1608, Y 18.2534, Z -1.3333, A 0.000, B 0.000, C 0.000 }
gfCNCPoint1[2305] = {X 472.5558, Y 16.5287, Z -1.3333, A 0.000, B 0.000, C 0.000 }
gfCNCPoint1[2306] = {X 473.0749, Y 15.0578, Z -1.3333, A 0.000, B 0.000, C 0.000 }
gfCNCPoint1[2307] = {X 473.7747, Y 13.6638, Z -1.3333, A 0.000, B 0.000, C 0.000 }
gfCNCPoint1[2308] = {X 474.6439, Y 12.3687, Z -1.3333, A 0.000, B 0.000, C 0.000 }
gfCNCPoint1[2309] = {X 475.6690, Y 11.1930, Z -1.3333, A 0.000, B 0.000, C 0.000 }
gfCNCPoint1[2310] = {X 476.7460, Y 10.2245, Z -1.3333, A 0.000, B 0.000, C 0.000 }
gfCNCPoint1[2311] = {X 477.9287, Y 9.3883, Z -1.3333, A 0.000, B 0.000, C 0.000 }
gfCNCPoint1[2312] = {X 479.2009, Y 8.6958, Z -1.3333, A 0.000, B 0.000, C 0.000 }
gfCNCPoint1[2313] = {X 480.5451, Y 8.1564, Z -1.3333, A 0.000, B 0.000, C 0.000 }
gfCNCPoint1[2314] = {X 481.9431, Y 7.7774, Z -1.3333, A 0.000, B 0.000, C 0.000 }
gfCNCPoint1[2315] = {X 484.0945, Y 7.4425, Z -1.3333, A 0.000, B 0.000, C 0.000 }
gfCNCPoint1[2316] = {X 486.2685, Y 7.3241, Z -1.3333, A 0.000, B 0.000, C 0.000 }
gfCNCPoint1[2317] = {X 486.9707, Y 7.3119, Z -1.3333, A 0.000, B 0.000, C 0.000 }
gfCNCPoint1[2318] = {X 502.2122, Y 7.3119, Z -1.3333, A 0.000, B 0.000, C 0.000 }
gfCNCPoint1[2319] = {X 502.7417, Y 7.3161, Z -1.3333, A 0.000, B 0.000, C 0.000 }
gfCNCPoint1[2320] = {X 503.6961, Y 7.4182, Z -1.3333, A 0.000, B 0.000, C 0.000 }
gfCNCPoint1[2321] = {X 504.6119, Y 7.7058, Z -1.3333, A 0.000, B 0.000, C 0.000 }
gfCNCPoint1[2322] = {X 505.4534, Y 8.1676, Z -1.3333, A 0.000, B 0.000, C 0.000 }
gfCNCPoint1[2323] = {X 506.1879, Y 8.7856, Z -1.3333, A 0.000, B 0.000, C 0.000 }
gfCNCPoint1[2324] = {X 506.7867, Y 9.5358, Z -1.3333, A 0.000, B 0.000, C 0.000 }
gfCNCPoint1[2325] = {X 507.2265, Y 10.3890, Z -1.3333, A 0.000, B 0.000, C 0.000 }
gfCNCPoint1[2326] = {X 507.4822, Y 11.2687, Z -1.3333, A 0.000, B 0.000, C 0.000 }
gfCNCPoint1[2327] = {X 507.5685, Y 12.1807, Z -1.3333, A 0.000, B 0.000, C 0.000 }
gfCNCPoint1[2328] = {X 507.5683, Y 13.0237, Z -1.3333, A 0.000, B 0.000, C 0.000 }
gfCNCPoint1[2329] = {X 507.4608, Y 13.9975, Z -1.3333, A 0.000, B 0.000, C 0.000 }
gfCNCPoint1[2330] = {X 507.1610, Y 14.9302, Z -1.3333, A 0.000, B 0.000, C 0.000 }
gfCNCPoint1[2331] = {X 506.6809, Y 15.7842, Z -1.3333, A 0.000, B 0.000, C 0.000 }
gfCNCPoint1[2332] = {X 506.0400, Y 16.5251, Z -1.3333, A 0.000, B 0.000, C 0.000 }
gfCNCPoint1[2333] = {X 506.0399, Y 40.6616, Z -1.3333, A 0.000, B 0.000, C 0.000 }
gfCNCPoint1[2334] = {X 506.6814, Y 41.4032, Z -1.3333, A 0.000, B 0.000, C 0.000 }
gfCNCPoint1[2335] = {X 507.1617, Y 42.2581, Z -1.3333, A 0.000, B 0.000, C 0.000 }
gfCNCPoint1[2336] = {X 507.4613, Y 43.1918, Z -1.3333, A 0.000, B 0.000, C 0.000 }
gfCNCPoint1[2337] = {X 507.5683, Y 44.1665, Z -1.3333, A 0.000, B 0.000, C 0.000 }
gfCNCPoint1[2338] = {X 507.5685, Y 45.0000, Z -1.3333, A 0.000, B 0.000, C 0.000 }
gfCNCPoint1[2339] = {X 507.4747, Y 45.9520, Z -1.3333, A 0.000, B 0.000, C 0.000 }
gfCNCPoint1[2340] = {X 507.1970, Y 46.8675, Z -1.3333, A 0.000, B 0.000, C 0.000 }
gfCNCPoint1[2341] = {X 506.7461, Y 47.7112, Z -1.3333, A 0.000, B 0.000, C 0.000 }
gfCNCPoint1[2342] = {X 506.1392, Y 48.4507, Z -1.3333, A 0.000, B 0.000, C 0.000 }
gfCNCPoint1[2343] = {X 505.3997, Y 49.0576, Z -1.3333, A 0.000, B 0.000, C 0.000 }
gfCNCPoint1[2344] = {X 504.5560, Y 49.5085, Z -1.3333, A 0.000, B 0.000, C 0.000 }
gfCNCPoint1[2345] = {X 503.6405, Y 49.7862, Z -1.3333, A 0.000, B 0.000, C 0.000 }
gfCNCPoint1[2346] = {X 502.6885, Y 49.8800, Z -1.3333, A 0.000, B 0.000, C 0.000 }
gfCNCPoint1[2347] = {X 496.2450, Y 49.8800, Z -1.3333, A 0.000, B 0.000, C 0.000 }
gfCNCPoint1[2348] = {X 495.2220, Y 49.7716, Z -1.3333, A 0.000, B 0.000, C 0.000 }
gfCNCPoint1[2349] = {X 494.2445, Y 49.4511, Z -1.3333, A 0.000, B 0.000, C 0.000 }
gfCNCPoint1[2350] = {X 493.3559, Y 48.9328, Z -1.3333, A 0.000, B 0.000, C 0.000 }
gfCNCPoint1[2351] = {X 492.5956, Y 48.2398, Z -1.3333, A 0.000, B 0.000, C 0.000 }
gfCNCPoint1[2352] = {X 491.9976, Y 47.4028, Z -1.3333, A 0.000, B 0.000, C 0.000 }
gfCNCPoint1[2353] = {X 491.5882, Y 46.4590, Z -1.3333, A 0.000, B 0.000, C 0.000 }
gfCNCPoint1[2354] = {X 491.4241, Y 45.7570, Z -1.3333, A 0.000, B 0.000, C 0.000 }
gfCNCPoint1[2355] = {X 491.3652, Y 45.0385, Z -1.3333, A 0.000, B 0.000, C 0.000 }
gfCNCPoint1[2356] = {X 491.3655, Y 44.1417, Z -1.3333, A 0.000, B 0.000, C 0.000 }
gfCNCPoint1[2357] = {X 491.4758, Y 43.1751, Z -1.3333, A 0.000, B 0.000, C 0.000 }
gfCNCPoint1[2358] = {X 491.7755, Y 42.2497, Z -1.3333, A 0.000, B 0.000, C 0.000 }
gfCNCPoint1[2359] = {X 492.2530, Y 41.4021, Z -1.3333, A 0.000, B 0.000, C 0.000 }
gfCNCPoint1[2360] = {X 492.8890, Y 40.6660, Z -1.3333, A 0.000, B 0.000, C 0.000 }
gfCNCPoint1[2361] = {X 492.8890, Y 35.0338, Z -1.3333, A 0.000, B 0.000, C 0.000 }
gfCNCPoint1[2362] = {X 491.0651, Y 35.0338, Z -1.3333, A 0.000, B 0.000, C 0.000 }
gfCNCPoint1[2363] = {X 487.0428, Y 42.8665, Z -1.3333, A 0.000, B 0.000, C 0.000 }
gfCNCPoint1[2364] = {X 487.1806, Y 43.5093, Z -1.3333, A 0.000, B 0.000, C 0.000 }
gfCNCPoint1[2365] = {X 487.2308, Y 44.1648, Z -1.3333, A 0.000, B 0.000, C 0.000 }
gfCNCPoint1[2366] = {X 487.2310, Y 45.0000, Z -1.3333, A 0.000, B 0.000, C 0.000 }
gfCNCPoint1[2367] = {X 487.1749, Y 45.7380, Z -1.3333, A 0.000, B 0.000, C 0.000 }
gfCNCPoint1[2368] = {X 487.0078, Y 46.4590, Z -1.3333, A 0.000, B 0.000, C 0.000 }
gfCNCPoint1[2369] = {X 486.5939, Y 47.4110, Z -1.3333, A 0.000, B 0.000, C 0.000 }
gfCNCPoint1[2370] = {X 485.9879, Y 48.2538, Z -1.3333, A 0.000, B 0.000, C 0.000 }
gfCNCPoint1[2371] = {X 485.2175, Y 48.9494, Z -1.3333, A 0.000, B 0.000, C 0.000 }
gfCNCPoint1[2372] = {X 484.3173, Y 49.4663, Z -1.3333, A 0.000, B 0.000, C 0.000 }
gfCNCPoint1[2373] = {X 483.3557, Y 49.7755, Z -1.3333, A 0.000, B 0.000, C 0.000 }
gfCNCPoint1[2374] = {X 482.3510, Y 49.8800, Z -1.3333, A 0.000, B 0.000, C 0.000 }
gfCNCPoint1[2375] = {X 480.2695, Y 49.8800, Z -1.3333, A 0.000, B 0.000, C 0.000 }
gfCNCPoint1[2376] = {X 480.2695, Y 49.4000, Z -1.3333, A 0.000, B 0.000, C 0.000 }
gfCNCPoint1[2377] = {X 475.7650, Y 49.4000, Z -1.3333, A 0.000, B 0.000, C 0.000 }
gfCNCPoint1[2378] = {X 474.7859, Y 49.2897, Z -1.3333, A 0.000, B 0.000, C 0.000 }
gfCNCPoint1[2379] = {X 473.8559, Y 48.9643, Z -1.3333, A 0.000, B 0.000, C 0.000 }
gfCNCPoint1[2380] = {X 473.0216, Y 48.4401, Z -1.3333, A 0.000, B 0.000, C 0.000 }
gfCNCPoint1[2381] = {X 472.3249, Y 47.7434, Z -1.3333, A 0.000, B 0.000, C 0.000 }
gfCNCPoint1[2382] = {X 471.8007, Y 46.9091, Z -1.3333, A 0.000, B 0.000, C 0.000 }
gfCNCPoint1[2383] = {X 471.4753, Y 45.9791, Z -1.3333, A 0.000, B 0.000, C 0.000 }
gfCNCPoint1[2384] = {X 471.3650, Y 45.0000, Z -1.3333, A 0.000, B 0.000, C 0.000 }
gfCNCPoint1[2385] = {X 471.3654, Y 44.1483, Z -1.3333, A 0.000, B 0.000, C 0.000 }
gfCNCPoint1[2386] = {X 471.4638, Y 43.2816, Z -1.3333, A 0.000, B 0.000, C 0.000 }
gfCNCPoint1[2387] = {X 471.7311, Y 42.4514, Z -1.3333, A 0.000, B 0.000, C 0.000 }
gfCNCPoint1[2388] = {X 472.1570, Y 41.6903, Z -1.3333, A 0.000, B 0.000, C 0.000 }
gfCNCPoint1[2389] = {X 472.7247, Y 41.0281, Z -1.3333, A 0.000, B 0.000, C 0.000 }
gfCNCPoint1[2390] = {X 473.4118, Y 40.4909, Z -1.3333, A 0.000, B 0.000, C 0.000 }
gfCNCPoint1[2391] = {X 474.1914, Y 40.0998, Z -1.3333, A 0.000, B 0.000, C 0.000 }
gfCNCPoint1[2392] = {X 478.1278, Y 32.3948, Z -1.3333, A 0.000, B 0.000, C 0.000 }
gfCNCPoint1[2393] = {X 476.8713, Y 31.5205, Z -1.3333, A 0.000, B 0.000, C 0.000 }
gfCNCPoint1[2394] = {X 475.7415, Y 30.4877, Z -1.3333, A 0.000, B 0.000, C 0.000 }
gfCNCPoint1[2395] = {X 474.7581, Y 29.3146, Z -1.3333, A 0.000, B 0.000, C 0.000 }
gfCNCPoint1[2396] = {X 473.9385, Y 28.0218, Z -1.3333, A 0.000, B 0.000, C 0.000 }
gfCNCPoint1[2397] = {X 473.2970, Y 26.6320, Z -1.3333, A 0.000, B 0.000, C 0.000 }
gfCNCPoint1[2398] = {X 472.8449, Y 25.1695, Z -1.3333, A 0.000, B 0.000, C 0.000 }
gfCNCPoint1[2399] = {X 472.5293, Y 23.4784, Z -1.3333, A 0.000, B 0.000, C 0.000 }
gfCNCPoint1[2400] = {X 472.3881, Y 21.7639, Z -1.3333, A 0.000, B 0.000, C 0.000 }
gfCNCPoint1[2401] = {X 472.4230, Y 20.0439, Z -1.3333, A 0.000, B 0.000, C 0.000 }
gfCNCPoint1[2402] = {X 472.6336, Y 18.3365, Z -1.3333, A 0.000, B 0.000, C 0.000 }
gfCNCPoint1[2403] = {X 473.0175, Y 16.6596, Z -1.3333, A 0.000, B 0.000, C 0.000 }
gfCNCPoint1[2404] = {X 473.5644, Y 15.1350, Z -1.3333, A 0.000, B 0.000, C 0.000 }
gfCNCPoint1[2405] = {X 474.3129, Y 13.6986, Z -1.3333, A 0.000, B 0.000, C 0.000 }
gfCNCPoint1[2406] = {X 475.2494, Y 12.3769, Z -1.3333, A 0.000, B 0.000, C 0.000 }
gfCNCPoint1[2407] = {X 476.3564, Y 11.1945, Z -1.3333, A 0.000, B 0.000, C 0.000 }
gfCNCPoint1[2408] = {X 477.6135, Y 10.1732, Z -1.3333, A 0.000, B 0.000, C 0.000 }
gfCNCPoint1[2409] = {X 478.9975, Y 9.3317, Z -1.3333, A 0.000, B 0.000, C 0.000 }
gfCNCPoint1[2410] = {X 480.4829, Y 8.6857, Z -1.3333, A 0.000, B 0.000, C 0.000 }
gfCNCPoint1[2411] = {X 482.0421, Y 8.2471, Z -1.3333, A 0.000, B 0.000, C 0.000 }
gfCNCPoint1[2412] = {X 484.1469, Y 7.9196, Z -1.3333, A 0.000, B 0.000, C 0.000 }
gfCNCPoint1[2413] = {X 486.2738, Y 7.8041, Z -1.3333, A 0.000, B 0.000, C 0.000 }
gfCNCPoint1[2414] = {X 486.9707, Y 7.7919, Z -1.3333, A 0.000, B 0.000, C 0.000 }
gfCNCPoint1[2415] = {X 502.2084, Y 7.7919, Z -1.3333, A 0.000, B 0.000, C 0.000 }
gfCNCPoint1[2416] = {X 502.7379, Y 7.7960, Z -1.3333, A 0.000, B 0.000, C 0.000 }
gfCNCPoint1[2417] = {X 503.7080, Y 7.9125, Z -1.3333, A 0.000, B 0.000, C 0.000 }
gfCNCPoint1[2418] = {X 504.6282, Y 8.2408, Z -1.3333, A 0.000, B 0.000, C 0.000 }
gfCNCPoint1[2419] = {X 505.4528, Y 8.7648, Z -1.3333, A 0.000, B 0.000, C 0.000 }
gfCNCPoint1[2420] = {X 506.1410, Y 9.4583, Z -1.3333, A 0.000, B 0.000, C 0.000 }
gfCNCPoint1[2421] = {X 506.6585, Y 10.2871, Z -1.3333, A 0.000, B 0.000, C 0.000 }
gfCNCPoint1[2422] = {X 506.9796, Y 11.2098, Z -1.3333, A 0.000, B 0.000, C 0.000 }
gfCNCPoint1[2423] = {X 507.0885, Y 12.1807, Z -1.3333, A 0.000, B 0.000, C 0.000 }
gfCNCPoint1[2424] = {X 507.0883, Y 13.0233, Z -1.3333, A 0.000, B 0.000, C 0.000 }
gfCNCPoint1[2425] = {X 506.9799, Y 13.9497, Z -1.3333, A 0.000, B 0.000, C 0.000 }
gfCNCPoint1[2426] = {X 506.6787, Y 14.8324, Z -1.3333, A 0.000, B 0.000, C 0.000 }
